 VAR PERSISTENT
//Conveyors Incoming 2000 (Purple line)
//Transport   
//----------------------------------------P2130--------------------------------------------------------------
cfgP2130IntlksArry: ARRAY [0..15] OF ST_CfgEvents := [
   (Description := 'Exit PE/Downstream MTR status' , DeviceLabel := '' , OKState := TRUE),   //DeviceLabel: Exit PE downstream
   (Description := 'System Interlocks' , DeviceLabel := '', OKState := TRUE, StopCode := E_StopCodes.SystemStop),
   13(())];
cfgP2130EvntsArry: ARRAY [0..15] OF ST_CfgEvents := [
   (Description := 'Jam Detected', DeviceLabel := '', LatchRequired := TRUE, OKState := FALSE, StopCode := E_StopCodes.ProductJam),   //DeviceLabel: Jam PE
   (),
   (Description := 'Disconnect', DeviceLabel := 'P2130', OKState := TRUE, StopCode := E_StopCodes.DisconnectState),   //DeviceLabel: Motor Disconnect
   (Description := 'System Fault', DeviceLabel := '', OKState := TRUE, FaultWarn:= TRUE, StopCode := E_StopCodes.SystemStop),
   (Description := 'RIO12182 Comm Fault', DeviceLabel := 'RIO12182', OKState := TRUE, FaultWarn:= TRUE, StopCode := E_StopCodes.FieldIOFLT),
   (Description := 'Power Transfer Raised', DeviceLabel := 'PX12151', OKState := TRUE, FaultWarn:= TRUE, StopCode := E_StopCodes.TransferLP),
   (Description := 'Motor Faulted', DeviceLabel := 'P2130', OKState := FALSE, StopCode := E_StopCodes.MotorOL),
   9(())];
//Transport
//----------------------------------------P2135--------------------------------------------------------------
cfgP2135IntlksArry: ARRAY [0..15] OF ST_CfgEvents := [
   (Description := 'Exit PE/Downstream MTR status' , DeviceLabel := '' , OKState := TRUE),   //DeviceLabel: Exit PE downstream
   (Description := 'System Interlocks' , DeviceLabel := '', OKState := TRUE, StopCode := E_StopCodes.SystemStop),
   11(())];
cfgP2135EvntsArry: ARRAY [0..15] OF ST_CfgEvents := [
   (Description := 'Jam Detected', DeviceLabel := '', LatchRequired := TRUE, OKState := FALSE, StopCode := E_StopCodes.ProductJam),   //DeviceLabel: Jam PE
   (),
   (Description := 'Disconnect', DeviceLabel := 'P2135', OKState := TRUE, StopCode := E_StopCodes.DisconnectState),   //DeviceLabel: Motor Disconnect
   (Description := 'System Fault', DeviceLabel := '', OKState := TRUE, FaultWarn:= TRUE, StopCode := E_StopCodes.SystemStop),
   (Description := 'RIO10161 Comm Fault', DeviceLabel := 'RIO10161', OKState := TRUE, FaultWarn:= TRUE, StopCode := E_StopCodes.FieldIOFLT),
   (Description := 'Motor Faulted', DeviceLabel := 'P2135', OKState := FALSE, StopCode := E_StopCodes.MotorOL),
   10(())];
//Transport
//----------------------------------------P2140--------------------------------------------------------------
cfgP2140IntlksArry: ARRAY [0..15] OF ST_CfgEvents := [
   (Description := 'Exit PE/Downstream MTR status' , DeviceLabel := '' , OKState := TRUE),   //DeviceLabel: Exit PE downstream
   (Description := 'System Interlocks' , DeviceLabel := '', OKState := TRUE, StopCode := E_StopCodes.SystemStop),
   (),
   (Description := 'GR2140-01 Auto', DeviceLabel := 'GR2140-01', OKState := TRUE, StopCode := E_StopCodes.DeviceNoInAuto),
   (Description := 'GR2140-02 Auto', DeviceLabel := 'GR2140-02', OKState := TRUE, StopCode := E_StopCodes.DeviceNoInAuto),
   (Description := 'PI2140-01 Auto', DeviceLabel := 'PI2140-01', OKState := TRUE, StopCode := E_StopCodes.DeviceNoInAuto),
   (Description := 'PL2140-01 Auto', DeviceLabel := 'PU2140-01', OKState := TRUE, StopCode := E_StopCodes.DeviceNoInAuto),
   9(())];
cfgP2140EvntsArry: ARRAY [0..15] OF ST_CfgEvents := [
   (Description := 'Jam Detected', DeviceLabel := '', LatchRequired := TRUE, OKState := FALSE, StopCode := E_StopCodes.ProductJam),   //DeviceLabel: Jam PE
   (),
   (Description := 'Disconnect', DeviceLabel := 'P2140', OKState := TRUE, StopCode := E_StopCodes.DisconnectState),   //DeviceLabel: Motor Disconnect
   (Description := 'System Fault', DeviceLabel := '', OKState := TRUE, FaultWarn:= TRUE, StopCode := E_StopCodes.SystemStop),
   (Description := 'RIO10161 Comm Fault', DeviceLabel := 'RIO10161', OKState := TRUE, FaultWarn:= TRUE, StopCode := E_StopCodes.FieldIOFLT),
   (Description := 'BCR_S2140_01 Comm Fault', DeviceLabel := 'BCR_S2140_01', OKState := TRUE, FaultWarn:= TRUE, StopCode := E_StopCodes.FieldIOFLT),
   (Description := 'Plow Jam', DeviceLabel := 'PL2140_01', OKState := TRUE, FaultWarn:= TRUE, StopCode := E_StopCodes.ProductJam),
   (Description := 'Motor Faulted', DeviceLabel := 'P2140', OKState := FALSE, StopCode := E_StopCodes.MotorOL),
   8(())];
//Transport
//----------------------------------------P2143--------------------------------------------------------------
cfgP2143IntlksArry: ARRAY [0..15] OF ST_CfgEvents := [
   (Description := 'Exit PE/Downstream MTR status' , DeviceLabel := '' , OKState := TRUE),   //DeviceLabel: Exit PE downstream
   (Description := 'System Interlocks' , DeviceLabel := '', OKState := TRUE, StopCode := E_StopCodes.SystemStop),
   13(())];
cfgP2143EvntsArry: ARRAY [0..15] OF ST_CfgEvents := [
   (Description := 'Jam Detected', DeviceLabel := '', LatchRequired := TRUE, OKState := FALSE, StopCode := E_StopCodes.ProductJam),   //DeviceLabel: Jam PE
   (),
   (Description := 'Disconnect', DeviceLabel := 'P2143', OKState := TRUE, StopCode := E_StopCodes.DisconnectState),   //DeviceLabel: Motor Disconnect
   (Description := 'System Fault', DeviceLabel := '', OKState := TRUE, FaultWarn:= TRUE, StopCode := E_StopCodes.SystemStop),
   (Description := 'RIO8171 Comm Fault', DeviceLabel := 'RIO8171', OKState := TRUE, FaultWarn:= TRUE, StopCode := E_StopCodes.FieldIOFLT),
   (Description := 'BCR_S2141_01 Comm Fault', DeviceLabel := 'BCR_S2141_011', OKState := TRUE, FaultWarn:= TRUE, StopCode := E_StopCodes.FieldIOFLT),
   (Description := 'Motor Faulted', DeviceLabel := 'P2143', OKState := FALSE, StopCode := E_StopCodes.MotorOL),
   9(())];
//Spiral
//----------------------------------------P2141--------------------------------------------------------------
cfgP2141IntlksArry: ARRAY [0..15] OF ST_CfgEvents := [
   (Description := 'Exit PE/Downstream MTR status' , DeviceLabel := '' , OKState := TRUE),   //DeviceLabel: Exit PE downstream
   (Description := 'System Interlocks' , DeviceLabel := '', OKState := TRUE, StopCode := E_StopCodes.SystemStop),
   14(())];
cfgP2141EvntsArry: ARRAY [0..15] OF ST_CfgEvents := [
   (Description := 'Jam Detected', DeviceLabel := '', LatchRequired := TRUE, OKState := FALSE, StopCode := E_StopCodes.ProductJam),   //DeviceLabel: Jam PE
   (),
   (Description := 'Disconnect', DeviceLabel := 'P2141', OKState := TRUE, StopCode := E_StopCodes.DisconnectState),   //DeviceLabel: Motor Disconnect
   (Description := 'System Fault', DeviceLabel := '', OKState := TRUE, FaultWarn:= TRUE, StopCode := E_StopCodes.SystemStop),
   (Description := 'RIO8171 Comm Fault', DeviceLabel := 'RIO8171', OKState := TRUE, FaultWarn:= TRUE, StopCode := E_StopCodes.FieldIOFLT),
   (Description := 'VFD State Not OK', DeviceLabel := 'P2141', OKState := TRUE, StopCode := E_StopCodes.VFD_Fault),
   10(())];
//Transport
//----------------------------------------P2142--------------------------------------------------------------
cfgP2142IntlksArry: ARRAY [0..15] OF ST_CfgEvents := [
   (Description := 'Exit PE/Downstream MTR status' , DeviceLabel := '' , OKState := TRUE),   //DeviceLabel: Exit PE downstream
   (Description := 'System Interlocks' , DeviceLabel := '', OKState := TRUE, StopCode := E_StopCodes.SystemStop),
   13(())];
cfgP2142EvntsArry: ARRAY [0..15] OF ST_CfgEvents := [
   (Description := 'Jam Detected', DeviceLabel := '', LatchRequired := TRUE, OKState := FALSE, StopCode := E_StopCodes.ProductJam),   //DeviceLabel: Jam PE
   (),
   (Description := 'Disconnect', DeviceLabel := 'P2142', OKState := TRUE, StopCode := E_StopCodes.DisconnectState),   //DeviceLabel: Motor Disconnect
   (Description := 'System Fault', DeviceLabel := '', OKState := TRUE, FaultWarn:= TRUE, StopCode := E_StopCodes.SystemStop),
   (Description := 'RIO8171 Comm Fault', DeviceLabel := 'RIO8171', OKState := TRUE, FaultWarn:= TRUE, StopCode := E_StopCodes.FieldIOFLT),
   (Description := 'Motor Faulted', DeviceLabel := 'P2142', OKState := FALSE, StopCode := E_StopCodes.MotorOL),
   10(())];
//Transport
//----------------------------------------P2145--------------------------------------------------------------
cfgP2145IntlksArry: ARRAY [0..15] OF ST_CfgEvents := [
   (Description := 'Exit PE/Downstream MTR status' , DeviceLabel := '' , OKState := TRUE),   //DeviceLabel: Exit PE downstream
   (Description := 'System Interlocks' , DeviceLabel := '', OKState := TRUE, StopCode := E_StopCodes.SystemStop),
   13(())];
cfgP2145EvntsArry: ARRAY [0..15] OF ST_CfgEvents := [
   (Description := 'Jam Detected', DeviceLabel := '', LatchRequired := TRUE, OKState := FALSE, StopCode := E_StopCodes.ProductJam),   //DeviceLabel: Jam PE
   (),
   (Description := 'Disconnect', DeviceLabel := 'P2145', OKState := TRUE, StopCode := E_StopCodes.DisconnectState),   //DeviceLabel: Motor Disconnect
   (Description := 'System Fault', DeviceLabel := '', OKState := TRUE, FaultWarn:= TRUE, StopCode := E_StopCodes.SystemStop),
   (Description := 'RIO2151 Comm Fault', DeviceLabel := 'RIO2151', OKState := TRUE, FaultWarn:= TRUE, StopCode := E_StopCodes.FieldIOFLT),
   (Description := 'Motor Faulted', DeviceLabel := 'P2145', OKState := FALSE, StopCode := E_StopCodes.MotorOL),
   10(())];
//Spiral
//----------------------------------------P2146--------------------------------------------------------------
cfgP2146IntlksArry: ARRAY [0..15] OF ST_CfgEvents := [
   (Description := 'Exit PE/Downstream MTR status' , DeviceLabel := '' , OKState := TRUE),   //DeviceLabel: Exit PE downstream
   (Description := 'System Interlocks' , DeviceLabel := '', OKState := TRUE, StopCode := E_StopCodes.SystemStop),
   (),
   12(())];
cfgP2146EvntsArry: ARRAY [0..15] OF ST_CfgEvents := [
   (Description := 'Jam Detected', DeviceLabel := '', LatchRequired := TRUE, OKState := FALSE, StopCode := E_StopCodes.ProductJam),   //DeviceLabel: Jam PE
   (),
   (Description := 'Disconnect', DeviceLabel := 'P2146', OKState := TRUE, StopCode := E_StopCodes.DisconnectState),   //DeviceLabel: Motor Disconnect
   (Description := 'System Fault', DeviceLabel := '', OKState := TRUE, FaultWarn:= TRUE, StopCode := E_StopCodes.SystemStop),
   (Description := 'RIO2151 Comm Fault', DeviceLabel := 'RIO2151', OKState := TRUE, FaultWarn:= TRUE, StopCode := E_StopCodes.FieldIOFLT),
   (Description := 'VFD State Not OK', DeviceLabel := 'P2146', OKState := TRUE, StopCode := E_StopCodes.VFD_Fault),
   10(())];
//Sorter
//----------------------------------------P2150--------------------------------------------------------------
cfgP2150IntlksArry: ARRAY [0..15] OF ST_CfgEvents := [
   (Description := 'Exit PE/Downstream MTR status' , DeviceLabel := '' , OKState := TRUE),   //DeviceLabel: Exit PE downstream
   (Description := 'System Interlocks' , DeviceLabel := '', OKState := TRUE, StopCode := E_StopCodes.SystemStop),
   (),
   (Description := 'GR2150-01 Auto', DeviceLabel := 'GR2150-01', OKState := TRUE, StopCode := E_StopCodes.DeviceNoInAuto),
   (Description := 'GR2150-02 Auto', DeviceLabel := 'GR2150-02', OKState := TRUE, StopCode := E_StopCodes.DeviceNoInAuto),
   (Description := 'PU2150-01 Auto', DeviceLabel := 'PU2150-01', OKState := TRUE, StopCode := E_StopCodes.DeviceNoInAuto),
   (Description := 'PU2150-02 Auto', DeviceLabel := 'PU2150-02', OKState := TRUE, StopCode := E_StopCodes.DeviceNoInAuto),
   (Description := 'PU2150-03 Auto', DeviceLabel := 'PU2150-03', OKState := TRUE, StopCode := E_StopCodes.DeviceNoInAuto),
   (Description := 'PU2150-04 Auto', DeviceLabel := 'PU2150-04', OKState := TRUE, StopCode := E_StopCodes.DeviceNoInAuto),
   7(())];
cfgP2150EvntsArry: ARRAY [0..15] OF ST_CfgEvents := [
   (Description := 'Jam Detected', DeviceLabel := '', LatchRequired := TRUE, OKState := FALSE, StopCode := E_StopCodes.ProductJam),   //DeviceLabel: Jam PE
   (),
   (Description := 'Disconnect', DeviceLabel := 'P2150', OKState := TRUE, StopCode := E_StopCodes.DisconnectState),   //DeviceLabel: Motor Disconnect
   (Description := 'System Fault', DeviceLabel := '', OKState := TRUE, FaultWarn:= TRUE, StopCode := E_StopCodes.SystemStop),
   (Description := 'RIO2151 Comm Fault', DeviceLabel := 'RIO2151', OKState := TRUE, FaultWarn:= TRUE, StopCode := E_StopCodes.FieldIOFLT),
   (Description := 'RIO3171 Comm Fault', DeviceLabel := 'RIO3171', OKState := TRUE, FaultWarn:= TRUE, StopCode := E_StopCodes.FieldIOFLT),
   (Description := 'RIO4141 Comm Fault', DeviceLabel := 'RIO4141', OKState := TRUE, FaultWarn:= TRUE, StopCode := E_StopCodes.FieldIOFLT),
   (Description := 'BCR_S2150_01 Comm Fault', DeviceLabel := 'BCR_S2150_01', OKState := TRUE, FaultWarn:= TRUE, StopCode := E_StopCodes.FieldIOFLT),
   (Description := 'Motor Faulted', DeviceLabel := 'P2150', OKState := FALSE, StopCode := E_StopCodes.MotorRunTO),
   7(())];
//Conveyors Incoming 3000 (Green line)
//Spiral
//----------------------------------------P3080--------------------------------------------------------------
cfgP3080IntlksArry: ARRAY [0..15] OF ST_CfgEvents := [
   (Description := 'Exit PE/Downstream MTR status' , DeviceLabel := '' , OKState := TRUE),   //DeviceLabel: Exit PE downstream
   (Description := 'System Interlocks' , DeviceLabel := '', OKState := TRUE, StopCode := E_StopCodes.SystemStop),
   (),
   12(())];
cfgP3080EvntsArry: ARRAY [0..15] OF ST_CfgEvents := [
   (Description := 'Jam Detected', DeviceLabel := '', LatchRequired := TRUE, OKState := FALSE, StopCode := E_StopCodes.ProductJam),   //DeviceLabel: Jam PE
   (),
   (Description := 'Disconnect', DeviceLabel := 'P3080', OKState := TRUE, StopCode := E_StopCodes.DisconnectState),   //DeviceLabel: Motor Disconnect
   (Description := 'System Fault', DeviceLabel := '', OKState := TRUE, FaultWarn:= TRUE, StopCode := E_StopCodes.SystemStop),
   (Description := 'RIO9191 Comm Fault', DeviceLabel := 'RIO9191', OKState := TRUE, FaultWarn:= TRUE, StopCode := E_StopCodes.FieldIOFLT),
   (Description := 'BCR_S2150_01 Comm Fault', DeviceLabel := 'BCR_S2150_01', OKState := TRUE, FaultWarn:= TRUE, StopCode := E_StopCodes.FieldIOFLT),
   (Description := 'Height Check', DeviceLabel := 'PE_12261', OKState := TRUE, FaultWarn:= TRUE, StopCode := E_StopCodes.OverHeightFLT),
   (Description := 'VFD State Not OK', DeviceLabel := 'P3080', OKState := TRUE, StopCode := E_StopCodes.VFD_Fault),
   8(())];
//Transport
//----------------------------------------P3085--------------------------------------------------------------
cfgP3085IntlksArry: ARRAY [0..15] OF ST_CfgEvents := [
   (Description := 'Exit PE/Downstream MTR status' , DeviceLabel := '' , OKState := TRUE),   //DeviceLabel: Exit PE downstream
   (Description := 'System Interlocks' , DeviceLabel := '', OKState := TRUE, StopCode := E_StopCodes.SystemStop),
   (),
   12(())];
cfgP3085EvntsArry: ARRAY [0..15] OF ST_CfgEvents := [
   (Description := 'Jam Detected', DeviceLabel := '', LatchRequired := TRUE, OKState := FALSE, StopCode := E_StopCodes.ProductJam),   //DeviceLabel: Jam PE
   (),
   (Description := 'Disconnect', DeviceLabel := 'P3085', OKState := TRUE, StopCode := E_StopCodes.DisconnectState),   //DeviceLabel: Motor Disconnect
   (Description := 'System Fault', DeviceLabel := '', OKState := TRUE, FaultWarn:= TRUE, StopCode := E_StopCodes.SystemStop),
   (Description := 'RIO12182 Comm Fault', DeviceLabel := 'RIO12182', OKState := TRUE, FaultWarn:= TRUE, StopCode := E_StopCodes.FieldIOFLT),
   (Description := 'Motor Faulted', DeviceLabel := 'P3085', OKState := FALSE, StopCode := E_StopCodes.MotorRunTO),
   10(())];
//Transport
//----------------------------------------P3090--------------------------------------------------------------
cfgP3090IntlksArry: ARRAY [0..15] OF ST_CfgEvents := [
   (Description := 'Exit PE/Downstream MTR status' , DeviceLabel := '' , OKState := TRUE),   //DeviceLabel: Exit PE downstream
   (Description := 'System Interlocks' , DeviceLabel := '', OKState := TRUE, StopCode := E_StopCodes.SystemStop),
   (),
   12(())];
cfgP3090EvntsArry: ARRAY [0..15] OF ST_CfgEvents := [
   (Description := 'Jam Detected', DeviceLabel := '', LatchRequired := TRUE, OKState := FALSE, StopCode := E_StopCodes.ProductJam),   //DeviceLabel: Jam PE
   (),
   (Description := 'Disconnect', DeviceLabel := 'P3090', OKState := TRUE, StopCode := E_StopCodes.DisconnectState),   //DeviceLabel: Motor Disconnect
   (Description := 'System Fault', DeviceLabel := '', OKState := TRUE, FaultWarn:= TRUE, StopCode := E_StopCodes.SystemStop),
   (Description := 'RIO12182 Comm Fault', DeviceLabel := 'RIO12182', OKState := TRUE, FaultWarn:= TRUE, StopCode := E_StopCodes.FieldIOFLT),
   (Description := 'Motor Faulted', DeviceLabel := 'P3090', OKState := FALSE, StopCode := E_StopCodes.MotorRunTO),
   10(())];
//Transport
//----------------------------------------P3095--------------------------------------------------------------
cfgP3095IntlksArry: ARRAY [0..15] OF ST_CfgEvents := [
   (Description := 'Exit PE/Downstream MTR status' , DeviceLabel := '' , OKState := TRUE),   //DeviceLabel: Exit PE downstream
   (Description := 'System Interlocks' , DeviceLabel := '', OKState := TRUE, StopCode := E_StopCodes.SystemStop),
   (),
   12(())];
cfgP3095EvntsArry: ARRAY [0..15] OF ST_CfgEvents := [
   (Description := 'Jam Detected', DeviceLabel := '', LatchRequired := TRUE, OKState := FALSE, StopCode := E_StopCodes.ProductJam),   //DeviceLabel: Jam PE
   (),
   (Description := 'Disconnect', DeviceLabel := 'P3095', OKState := TRUE, StopCode := E_StopCodes.DisconnectState),   //DeviceLabel: Motor Disconnect
   (Description := 'System Fault', DeviceLabel := '', OKState := TRUE, FaultWarn:= TRUE, StopCode := E_StopCodes.SystemStop),
   (Description := 'RIO12182 Comm Fault', DeviceLabel := 'RIO12182', OKState := TRUE, FaultWarn:= TRUE, StopCode := E_StopCodes.FieldIOFLT),
   (Description := 'Power Transfer Raised', DeviceLabel := 'PX12251', OKState := TRUE, FaultWarn:= TRUE, StopCode := E_StopCodes.TransferLP),
   (Description := 'Motor Faulted', DeviceLabel := 'P3095', OKState := FALSE, StopCode := E_StopCodes.MotorOL),
   9(())];
P2141_Velocity: INT := 1800;
P2146_Velocity: INT := 1800;
P3080_Velocity: INT := 1800;
END_VAR

ResetAllDrives := System.Cnvyr_Reset; //Reset For VFD
//EAP
GVL_IO.To205_P2130_IsRunning := P2130_Status.Sts_IsRunning;
GVL_IO.To205_P3095_SendingProduct := P3095_Status.Sts_IsRunning OR Photoeyes.PE_12091.Out OR Photoeyes.PE_12181.Out;

//Conveyors Incoming 2000 (Purple line)
//Transport
//----------------------------------------P2130--------------------------------------------------------------
P2130_StatePB.AutoPB := System.Cnvyr_Auto;
P2130_StatePB.ManPB := System.Cnvyr_Manual;
P2130_StatePB.ResetPB := System.Cnvyr_Reset;
P2130_StatePB.OfflinePB := System.Cnvyr_Offline;
P2130SleepWakeTrig[1] := GVL_IO.From205_P2125_SendingProduct; //EAP Wakeup bits 

// Initialize the Equipment Type
P2130_Status.Sts_EquipmentState.EquipType := E_EquipType.Conveyor;

// Interlocks
//P2130.In_EquipIntlks.2:=
//Events
P2130.In_EquipEvents.2:= GVL_IO.DS_P2130;
P2130.In_EquipEvents.3:= System.SysEventsAllOk;
P2130.In_EquipEvents.4:= NOT CommStatus.RIO12182_CommFault.Out;
P2130.In_EquipEvents.5:= ProxSensors.PX_12151_Extended.Out;
P2130.In_EquipEvents.6:= NOT GVL_IO.P2130_Faulted;

// Function Call
P2130(
   In_p_EquipStatePB:= P2130_StatePB,
   In_P_ConvReqRun:= TRUE,
   In_ConvDwnStrmMtrStatus:=  P2135_Status.Sts_IsRunning,
   In_ConvCrntExitPhotoEye:=  Photoeyes.PE_12171.Out,
   In_SimActive:= System.Sys_SimActive,
   In_EquipInit:= GVL_IO.INIT,
   In_WakeSlpTrigArry:= P2130SleepWakeTrig,
   Cfg_EquipIndex := GVL_EquipArrays.nEquipIndex,
   Cfg_EquipLabel := cfgP2130Label,
   Cfg_EquipDefState:= System.ConvDefaultState,
   Cfg_EquipIntlksArry:= cfgP2130IntlksArry,
   Cfg_EquipEvntsArry:= cfgP2130EvntsArry,
   cfg_JamDetectTime:= cfgP2130JamDetectTime,
   Cfg_UseSleepTmr := TRUE,
   Cfg_UseStartUpDelay := TRUE,
   Cfg_StartUpDelayTime := T#500MS,
   Cfg_SleepWaitTime:= cfgP2130SleepTime,
   Sts_EquipState := P2130_Status,
   Out_ConvCrntMtr => GVL_IO.P2130_RUN);

P2130_Status.Sts_IsRunning := GVL_IO.P2130_RUN;

//Transport
//----------------------------------------P2135--------------------------------------------------------------
P2135_StatePB.AutoPB := System.Cnvyr_Auto;
P2135_StatePB.ManPB := System.Cnvyr_Manual;
P2135_StatePB.ResetPB := System.Cnvyr_Reset;
P2135_StatePB.OfflinePB := System.Cnvyr_Offline;
P2135SleepWakeTrig[1] := Photoeyes.PE_12171.Out;
//EAP from 3rd floor

// Initialize the Equipment Type
P2135_Status.Sts_EquipmentState.EquipType := E_EquipType.Conveyor;

// Interlocks
//P2135.In_EquipIntlks.2:=
//Events
P2135.In_EquipEvents.2:= GVL_IO.DS_P2135;
P2135.In_EquipEvents.3:= System.SysEventsAllOk;
P2135.In_EquipEvents.4:= NOT CommStatus.RIO10161_CommFault.Out;
P2135.In_EquipEvents.5:= NOT GVL_IO.P2135_Faulted;

// Function Call
P2135(
   In_p_EquipStatePB:= P2135_StatePB,
   In_P_ConvReqRun:= TRUE,
   In_ConvDwnStrmMtrStatus:= P2140_Status.Sts_IsRunning,
   In_ConvCrntExitPhotoEye:=  Photoeyes.PE_10291.Out,
   In_SimActive:= System.Sys_SimActive,
   In_EquipInit:= GVL_IO.INIT,
   In_WakeSlpTrigArry:= P2135SleepWakeTrig,
   Cfg_EquipIndex := GVL_EquipArrays.nEquipIndex,
   Cfg_EquipLabel := cfgP2135Label,
   Cfg_EquipDefState:= System.ConvDefaultState,
   Cfg_EquipIntlksArry:= cfgP2135IntlksArry,
   Cfg_EquipEvntsArry:= cfgP2135EvntsArry,
   cfg_JamDetectTime:= cfgP2135JamDetectTime,
   Cfg_UseSleepTmr := TRUE,
   Cfg_UseStartUpDelay := TRUE,
   Cfg_StartUpDelayTime := T#500MS,
   Cfg_SleepWaitTime:= cfgP2135SleepTime,
   Sts_EquipState := P2135_Status,
   Out_ConvCrntMtr => GVL_IO.P2135_RUN);

P2135_Status.Sts_IsRunning := GVL_IO.P2135_RUN;
//Transport
//----------------------------------------P2140--------------------------------------------------------------
P2140_StatePB.AutoPB := System.Cnvyr_Auto;
P2140_StatePB.ManPB := System.Cnvyr_Manual;
P2140_StatePB.ResetPB := System.Cnvyr_Reset;
P2140_StatePB.OfflinePB := System.Cnvyr_Offline;
P2140SleepWakeTrig[1] := Photoeyes.PE_10291.Out;
P2140SleepWakeTrig[2] := Photoeyes.PE_12171.Out;

// Initialize the Equipment Type
P2140_Status.Sts_EquipmentState.EquipType := E_EquipType.Conveyor;

// Interlocks
P2140.In_EquipIntlks.3:= Solenoids.GR2140_01_Status.Sts_EquipmentState.StsAuto;
P2140.In_EquipIntlks.4:= Solenoids.GR2140_02_Status.Sts_EquipmentState.StsAuto;
P2140.In_EquipIntlks.5:= Solenoids.PI2140_01_Status.Sts_EquipmentState.StsAuto;
P2140.In_EquipIntlks.6:= Solenoids.PL2140_01_Status.Sts_EquipmentState.StsAuto; 
//Events
P2140.In_EquipEvents.2:= GVL_IO.DS_P2140;
P2140.In_EquipEvents.3:= System.SysEventsAllOk;
P2140.In_EquipEvents.4:= NOT CommStatus.RIO10161_CommFault.Out;
P2140.In_EquipEvents.5:= NOT CommStatus.BCR_S2140_01_CommFault.Out;
P2140.In_EquipEvents.6:= FALSE;//Photoeyes.PE_10151.JamDetected AND Not Solenoids.PL2140_01.Out_ExtendCrntSV;
P2140.In_EquipEvents.7:= NOT GVL_IO.P2140_Faulted;
P2140.In_EquipEvents.8:= Photoeyes.PE_10151.JamDetected; 

// Function Call
P2140(
   In_p_EquipStatePB:= P2140_StatePB,
   In_P_ConvReqRun:= TRUE,
   In_ConvDwnStrmMtrStatus:= P2145_Status.Sts_IsRunning,
   In_ConvCrntExitPhotoEye:= Photoeyes.PE_10091.Out,
   In_SimActive:= System.Sys_SimActive,
   In_EquipInit:= GVL_IO.INIT,
   In_WakeSlpTrigArry:= P2140SleepWakeTrig,
   Cfg_EquipIndex := GVL_EquipArrays.nEquipIndex,
   Cfg_EquipLabel := cfgP2140Label,
   Cfg_EquipDefState:= System.ConvDefaultState,
   Cfg_EquipIntlksArry:= cfgP2140IntlksArry,
   Cfg_EquipEvntsArry:= cfgP2140EvntsArry,
   cfg_JamDetectTime:= cfgP2140JamDetectTime,
   Cfg_UseSleepTmr := TRUE,
   Cfg_UseStartUpDelay := TRUE,
   Cfg_StartUpDelayTime := T#500MS,
   Cfg_SleepWaitTime:= cfgP2140SleepTime,
   Sts_EquipState := P2140_Status,
   Out_ConvCrntMtr => GVL_IO.P2140_RUN);

P2140_Status.Sts_IsRunning := GVL_IO.P2140_RUN;
//Transport
//----------------------------------------P2143--------------------------------------------------------------
P2143_StatePB.AutoPB := System.Cnvyr_Auto;
P2143_StatePB.ManPB := System.Cnvyr_Manual;
P2143_StatePB.ResetPB := System.Cnvyr_Reset;
P2143_StatePB.OfflinePB := System.Cnvyr_Offline;
P2143SleepWakeTrig[1] := Photoeyes.PE_10291.Out;
P2143SleepWakeTrig[2] := Photoeyes.PE_12171.Out;

// Initialize the Equipment Type
P2143_Status.Sts_EquipmentState.EquipType := E_EquipType.Conveyor;

// Interlocks
//P2143.In_EquipIntlks.2:= 
//Events
P2143.In_EquipEvents.2:= GVL_IO.DS_P2143;
P2143.In_EquipEvents.3:= System.SysEventsAllOk;
P2143.In_EquipEvents.4:= NOT CommStatus.RIO8171_CommFault.Out;
P2143.In_EquipEvents.5:= NOT CommStatus.BCR_S2141_01_CommFault.Out;
P2143.In_EquipEvents.6:= NOT GVL_IO.P2143_Faulted;

// Function Call
P2143(
   In_p_EquipStatePB:= P2143_StatePB,
   In_P_ConvReqRun:= TRUE,
   In_ConvDwnStrmMtrStatus:=  P2141_VFD.IsRunning,
   In_ConvCrntExitPhotoEye:= Photoeyes.PE_8161.Out,
   In_SimActive:= System.Sys_SimActive,
   In_EquipInit:= GVL_IO.INIT,
   In_WakeSlpTrigArry:= P2143SleepWakeTrig,
   Cfg_EquipIndex := GVL_EquipArrays.nEquipIndex,
   Cfg_EquipLabel := cfgP2143Label,
   Cfg_EquipDefState:= System.ConvDefaultState,
   Cfg_EquipIntlksArry:= cfgP2143IntlksArry,
   Cfg_EquipEvntsArry:= cfgP2143EvntsArry,
   cfg_JamDetectTime:= cfgP2143JamDetectTime,
   Cfg_UseSleepTmr := TRUE,
   Cfg_UseStartUpDelay := TRUE,
   Cfg_StartUpDelayTime := T#500MS,
   Cfg_SleepWaitTime:= cfgP2143SleepTime,
   Sts_EquipState := P2143_Status,
   Out_ConvCrntMtr => GVL_IO.P2143_RUN);

P2143_Status.Sts_IsRunning := GVL_IO.P2143_RUN;
//Spiral
//----------------------------------------P2141--------------------------------------------------------------
P2141_StatePB.AutoPB := System.Cnvyr_Auto;
P2141_StatePB.ManPB := System.Cnvyr_Manual;
P2141_StatePB.ResetPB := System.Cnvyr_Reset;
P2141_StatePB.OfflinePB := System.Cnvyr_Offline;
P2141SleepWakeTrig[1] := Photoeyes.PE_8161.Out;
P2141SleepWakeTrig[2] := Photoeyes.PE_10151.Out;

// Initialize the Equipment Type
P2141_Status.Sts_EquipmentState.EquipType := E_EquipType.Conveyor;

// Interlocks
// Interlock the full for a stop only when the warning is on for the downstream conveyor
P2141.In_EquipIntlks.2:= Photoeyes.PE_8131.Out_OnOffFltrd AND P2142.Sts_WarnsArry[6].Status;

//Events
P2141.In_EquipEvents.2:= GVL_IO.DS_P2141;
P2141.In_EquipEvents.3:= System.SysEventsAllOk;
P2141.In_EquipEvents.4:= NOT CommStatus.RIO8171_CommFault.Out;
P2141.In_EquipEvents.5:= NOT P2141_VFD.IsFaulted;

// Function Call
P2141(
   In_p_EquipStatePB:= P2141_StatePB,
   In_P_ConvReqRun:= TRUE,
   In_ConvDwnStrmMtrStatus:= P2142_Status.Sts_IsRunning AND NOT P2142.Sts_WarnsArry[6].Status,
   In_ConvCrntExitPhotoEye:= Photoeyes.PE_8131.Out,
   In_SimActive:= System.Sys_SimActive,
   In_EquipInit:= GVL_IO.INIT,
   In_WakeSlpTrigArry:= P2141SleepWakeTrig,
   Cfg_EquipIndex := GVL_EquipArrays.nEquipIndex,
   Cfg_EquipLabel := cfgP2141Label,
   Cfg_EquipDefState:= System.ConvDefaultState,
   Cfg_EquipIntlksArry:= cfgP2141IntlksArry,
   Cfg_EquipEvntsArry:= cfgP2141EvntsArry,
   cfg_JamDetectTime:= cfgP2141JamDetectTime,
   Cfg_UseSleepTmr := TRUE,
   Cfg_UseStartUpDelay := TRUE,
   Cfg_StartUpDelayTime := T#500MS,
   Cfg_SleepWaitTime:= cfgP2141SleepTime,
   Sts_EquipState := P2141_Status);

//Motor Control
P2141_VFD(
   RunVelocity := P2141_Velocity,
   VelocityThreshold := DefaultVelocityThreshold,
   Reset := ResetAllDrives,
   RunRequest := (P2141.Out_ConvCrntMtr OR Test_VFD_P2141));
P2141_Status.Sts_IsRunning := P2141_VFD.IsRunning;
//Transport
//----------------------------------------P2142--------------------------------------------------------------
P2142_StatePB.AutoPB := System.Cnvyr_Auto;
P2142_StatePB.ManPB := System.Cnvyr_Manual;
P2142_StatePB.ResetPB := System.Cnvyr_Reset;
P2142_StatePB.OfflinePB := System.Cnvyr_Offline;
P2142SleepWakeTrig[1] := Photoeyes.PE_8131.Out;
P2142SleepWakeTrig[2] := Photoeyes.PE_8161.Out;

// Initialize the Equipment Type
P2142_Status.Sts_EquipmentState.EquipType := E_EquipType.Conveyor;

// Interlocks
//P2142.In_EquipIntlks.2:= Photoeyes.PE_8141.Out_OnFltrd;

//Events
P2142.In_EquipEvents.2:= GVL_IO.DS_P2142;
P2142.In_EquipEvents.3:= System.SysEventsAllOk;
P2142.In_EquipEvents.4:= NOT CommStatus.RIO8171_CommFault.Out;
P2142.In_EquipEvents.5:= NOT GVL_IO.P2142_Faulted;
P2142.In_EquipEvents.6 := Photoeyes.PE_8141.Out_OnOffFltrd AND Photoeyes.PE_8191.Out_OnOffFltrd;

// Function Call
P2142(
   In_p_EquipStatePB:= P2142_StatePB,
   In_P_ConvReqRun:= TRUE,
   In_ConvDwnStrmMtrStatus:= TRUE,
   In_ConvCrntExitPhotoEye:=  FALSE,
   Cfg_ConvType:= E_ConvType.end,
   In_SimActive:= System.Sys_SimActive,
   In_EquipInit:= GVL_IO.INIT,
   In_WakeSlpTrigArry:= P2142SleepWakeTrig,
   Cfg_EquipIndex := GVL_EquipArrays.nEquipIndex,
   Cfg_EquipLabel := cfgP2142Label,
   Cfg_EquipDefState:= System.ConvDefaultState,
   Cfg_EquipIntlksArry:= cfgP2142IntlksArry,
   Cfg_EquipEvntsArry:= cfgP2142EvntsArry,
   cfg_JamDetectTime:= cfgP2142JamDetectTime,
   Cfg_UseSleepTmr := TRUE,
   Cfg_UseStartUpDelay := TRUE,
   Cfg_StartUpDelayTime := T#500MS,
   Cfg_SleepWaitTime:= cfgP2142SleepTime,
   Sts_EquipState := P2142_Status,
   Out_ConvCrntMtr => GVL_IO.P2142_RUN);

P2142_Status.Sts_IsRunning := GVL_IO.P2142_RUN;
//Transport
//----------------------------------------P2145--------------------------------------------------------------
P2145_StatePB.AutoPB := System.Cnvyr_Auto;
P2145_StatePB.ManPB := System.Cnvyr_Manual;
P2145_StatePB.ResetPB := System.Cnvyr_Reset;
P2145_StatePB.OfflinePB := System.Cnvyr_Offline;
P2145SleepWakeTrig[1] := PhotoEyes.PE_10091.Out_OffFltrd;
P2145SleepWakeTrig[2] := PhotoEyes.PE_10291.Out_OffFltrd;

// Initialize the Equipment Type
P2145_Status.Sts_EquipmentState.EquipType := E_EquipType.Conveyor;

// Interlocks
//P2145.In_EquipIntlks.2:= 
//Events
P2145.In_EquipEvents.2:= GVL_IO.DS_P2145;
P2145.In_EquipEvents.3:= System.SysEventsAllOk;
P2145.In_EquipEvents.4:= NOT CommStatus.RIO2151_CommFault.Out;
P2145.In_EquipEvents.5:= NOT GVL_IO.P2145_Faulted;

// Function Call
P2145(
   In_p_EquipStatePB:= P2145_StatePB,
   In_P_ConvReqRun:= TRUE,
   In_ConvDwnStrmMtrStatus:=  P2146_VFD.IsRunning,
   In_ConvCrntExitPhotoEye:=  PhotoEyes.PE_2231.Out,
   In_SimActive:= System.Sys_SimActive,
   In_EquipInit:= GVL_IO.INIT,
   In_WakeSlpTrigArry:= P2145SleepWakeTrig,
   Cfg_EquipIndex := GVL_EquipArrays.nEquipIndex,
   Cfg_EquipLabel := cfgP2145Label,
   Cfg_EquipDefState:= System.ConvDefaultState,
   Cfg_EquipIntlksArry:= cfgP2145IntlksArry,
   Cfg_EquipEvntsArry:= cfgP2145EvntsArry,
   cfg_JamDetectTime:= cfgP2145JamDetectTime,
   Cfg_UseSleepTmr := TRUE,
   Cfg_UseStartUpDelay := TRUE,
   Cfg_StartUpDelayTime := T#500MS,
   Cfg_SleepWaitTime:= cfgP2145SleepTime,
   Sts_EquipState := P2145_Status,
   Out_ConvCrntMtr => GVL_IO.P2145_RUN);

P2145_Status.Sts_IsRunning := GVL_IO.P2145_RUN;
//Spiral
//----------------------------------------P2146--------------------------------------------------------------
P2146_StatePB.AutoPB := System.Cnvyr_Auto;
P2146_StatePB.ManPB := System.Cnvyr_Manual;
P2146_StatePB.ResetPB := System.Cnvyr_Reset;
P2146_StatePB.OfflinePB := System.Cnvyr_Offline;
P2146SleepWakeTrig[1] := PhotoEyes.PE_2231.Out_OffFltrd;
P2145SleepWakeTrig[2] := PhotoEyes.PE_10091.Out_OffFltrd;

// Initialize the Equipment Type
P2146_Status.Sts_EquipmentState.EquipType := E_EquipType.Conveyor;

// Interlocks
P2146.In_EquipIntlks.2:= Photoeyes.PE_2101.Out_OnOffFltrd AND Photoeyes.PE_2201.Out_OnOffFltrd;
//Events
P2146.In_EquipEvents.2:= GVL_IO.DS_P2146;
P2146.In_EquipEvents.3:= System.SysEventsAllOk;
P2146.In_EquipEvents.4:= NOT CommStatus.RIO2151_CommFault.Out;
P2146.In_EquipEvents.5:= NOT P2146_VFD.IsFaulted;

// Function Call
P2146(
   In_p_EquipStatePB:= P2146_StatePB,
   In_P_ConvReqRun:= TRUE,
   In_ConvDwnStrmMtrStatus:= P2150_Status.Sts_IsRunning,
   In_ConvCrntExitPhotoEye:= Photoeyes.PE_2201.Out_OffFltrd,
   In_SimActive:= System.Sys_SimActive,
   In_EquipInit:= GVL_IO.INIT,
   In_WakeSlpTrigArry:= P2146SleepWakeTrig,
   Cfg_EquipIndex := GVL_EquipArrays.nEquipIndex,
   Cfg_EquipLabel := cfgP2146Label,
   Cfg_EquipDefState:= System.ConvDefaultState,
   Cfg_EquipIntlksArry:= cfgP2146IntlksArry,
   Cfg_EquipEvntsArry:= cfgP2146EvntsArry,
   cfg_JamDetectTime:= cfgP2146JamDetectTime,
   Cfg_UseSleepTmr := TRUE,
   Cfg_UseStartUpDelay := FALSE,
   Cfg_SleepWaitTime:= cfgP2146SleepTime,
   Sts_EquipState := P2146_Status);

//Motor Control
P2146_VFD(
   RunVelocity := P2146_Velocity,
   VelocityThreshold := DefaultVelocityThreshold,
   Reset := ResetAllDrives,
   RunRequest := (P2146.Out_ConvCrntMtr OR Test_VFD_P2146));
P2146_Status.Sts_IsRunning := P2146_VFD.IsRunning;
//Sorter
//----------------------------------------P2150--------------------------------------------------------------
P2150_StatePB.AutoPB := System.Cnvyr_Auto OR GVL_IO.PB_RemoteReset_3211;
P2150_StatePB.ManPB := System.Cnvyr_Manual;
P2150_StatePB.ResetPB := System.Cnvyr_Reset OR GVL_IO.PB_RemoteReset_3211;
P2150_StatePB.OfflinePB := System.Cnvyr_Offline;
P2150SleepWakeTrig[1] := PhotoEyes.PE_2201.Out_OffFltrd;
P2150SleepWakeTrig[2] := PhotoEyes.PE_2231.Out_OffFltrd;
P2150SleepWakeTrig[3] := PhotoEyes.PE_2131.Out_OffFltrd;
P2150SleepWakeTrig[4] := PhotoEyes.PE_2101.Out_OffFltrd;


// Initialize the Equipment Type
P2150_Status.Sts_EquipmentState.EquipType := E_EquipType.Conveyor;

// Interlocks
P2150.In_EquipIntlks.2:= Singulation_Control.SortSingulation_P2150.Out_Ready;
P2150.In_EquipIntlks.3:= Solenoids.GR2150_01_Status.Sts_EquipmentState.StsAuto;
P2150.In_EquipIntlks.4:= Solenoids.PI2150_01_Status.Sts_EquipmentState.StsAuto;
P2150.In_EquipIntlks.5:= Solenoids.PU2150_01_Status.Sts_EquipmentState.StsAuto;
P2150.In_EquipIntlks.6:= Solenoids.PU2150_02_Status.Sts_EquipmentState.StsAuto;
P2150.In_EquipIntlks.7:= Solenoids.PU2150_03_Status.Sts_EquipmentState.StsAuto;
P2150.In_EquipIntlks.8:= Solenoids.PU2150_04_Status.Sts_EquipmentState.StsAuto;
P2150.In_EquipIntlks.9:= Sorter.aSorterDiverts_P2150[1].Full;
P2150.In_EquipIntlks.10:= Sorter.aSorterDiverts_P2150[2].Full;
P2150.In_EquipIntlks.11:= Sorter.aSorterDiverts_P2150[3].Full;
P2150.In_EquipIntlks.12:= Sorter.aSorterDiverts_P2150[4].Full;

//Events
P2150.In_EquipEvents.2:= GVL_IO.DS_P2150;
P2150.In_EquipEvents.3:= System.SysEventsAllOk;
P2150.In_EquipEvents.4:= NOT CommStatus.RIO2151_CommFault.Out;
P2150.In_EquipEvents.5:= NOT CommStatus.RIO3171_CommFault.Out;
P2150.In_EquipEvents.6:= NOT CommStatus.RIO4141_CommFault.Out;
P2150.In_EquipEvents.7:= NOT CommStatus.BCR_S2150_01_CommFault.Out;
P2150.In_EquipEvents.8:= NOT GVL_IO.P2150_Faulted;
P2150.In_EquipEvents.9:= Photoeyes.PE_2101.Out_OnOffFltrd;
P2150.In_EquipEvents.10:= Sorter.aSorterDiverts_P2150[1].Jammed;
P2150.In_EquipEvents.11:= Sorter.aSorterDiverts_P2150[2].Jammed;
P2150.In_EquipEvents.12:= Sorter.aSorterDiverts_P2150[3].Jammed;
P2150.In_EquipEvents.13:= Sorter.aSorterDiverts_P2150[4].Jammed;

// Function Call
P2150(
	In_p_EquipStatePB:= P2150_StatePB,
	In_P_ConvReqRun:= TRUE,
	In_ConvCrntExitPhotoEye:= PhotoEyes.PE_4161.Out,
	Cfg_ConvType:= E_ConvType.end,
	In_SimActive:= System.Sys_SimActive,
	In_EquipInit:= GVL_IO.INIT,
	In_WakeSlpTrigArry:= P2150SleepWakeTrig,
	Cfg_EquipIndex := GVL_EquipArrays.nEquipIndex,
	Cfg_EquipLabel := cfgP2150Label,
	Cfg_EquipDefState:= System.ConvDefaultState,
	Cfg_EquipIntlksArry:= cfgP2150IntlksArry,
	Cfg_EquipEvntsArry:= cfgP2150EvntsArry,
	cfg_JamDetectTime:= T#2S,
	Cfg_UseSleepTmr := TRUE,
	Cfg_SleepWaitTime:= cfgP2150SleepTime,
	Sts_EquipState := P2150_Status,
	Out_ConvCrntMtr => GVL_IO.P2150_RUN);

P2150_Status.Sts_IsRunning := GVL_IO.P2150_RUN;
//Conveyors Incoming 3000 (Green line)
//Spiral
//----------------------------------------P3080--------------------------------------------------------------
P3080_StatePB.AutoPB := System.Cnvyr_Auto OR GVL_IO.PB_RemoteReset_8251;
P3080_StatePB.ManPB := System.Cnvyr_Manual;
P3080_StatePB.ResetPB := System.Cnvyr_Reset OR GVL_IO.PB_RemoteReset_8251;
P3080_StatePB.OfflinePB := System.Cnvyr_Offline;
P3080_ResetWakeTmr(IN:= GVL_IO.PB_RemoteReset_8251, PT:= T#3S, Q=> );
P3080SleepWakeTrig[1] := P3080_ResetWakeTmr.Q; //Reset Button
P3080SleepWakeTrig[2] := Photoeyes.PE_9141.Out; //Photo Eye
P3080SleepWakeTrig[3] := Photoeyes.PE_9161.Out; //Photo Eye
P3080SleepWakeTrig[4] := Photoeyes.PE_9191.Out; //Photo Eye

// Initialize the Equipment Type
P3080_Status.Sts_EquipmentState.EquipType := E_EquipType.Conveyor;

// Interlocks
//P3080.In_EquipIntlks.2:= 
//Events
P3080.In_EquipEvents.2:= GVL_IO.DS_P3080;
P3080.In_EquipEvents.3:= System.SysEventsAllOk;
P3080.In_EquipEvents.4:= NOT CommStatus.RIO9191_CommFault.Out;
P3080.In_EquipEvents.5:= NOT CommStatus.BCR_S2150_01_CommFault.Out;
P3080.In_EquipEvents.6:= Photoeyes.PE_9221.Out;
P3080.In_EquipEvents.7:= NOT P3080_VFD.IsFaulted;

// Function Call
P3080(
   In_p_EquipStatePB:= P3080_StatePB,
   In_P_ConvReqRun:= TRUE,
   In_ConvDwnStrmMtrStatus:= P3085_Status.Sts_IsRunning,
   In_ConvCrntExitPhotoEye:= Photoeyes.PE_9191.Out, 
   In_SimActive:= System.Sys_SimActive,
   In_EquipInit:= GVL_IO.INIT,
   In_WakeSlpTrigArry:= P3080SleepWakeTrig,
   Cfg_EquipIndex := GVL_EquipArrays.nEquipIndex,
   Cfg_EquipLabel := cfgP3080Label,
   Cfg_EquipDefState:= System.ConvDefaultState,
   Cfg_EquipIntlksArry:= cfgP3080IntlksArry,
   Cfg_EquipEvntsArry:= cfgP3080EvntsArry,
   cfg_JamDetectTime:= cfgP3080JamDetectTime,
   Cfg_UseSleepTmr := TRUE,
   Cfg_UseStartUpDelay := TRUE,
   Cfg_StartUpDelayTime := T#500MS,
   Cfg_SleepWaitTime:= cfgP3080SleepTime,
   Sts_EquipState := P3080_Status);

//Motor Control
P3080_VFD(
   RunVelocity := P3080_Velocity,
   VelocityThreshold := DefaultVelocityThreshold,
   Reset := ResetAllDrives,
   RunRequest := (P3080.Out_ConvCrntMtr OR Test_VFD_P3080));
P3080_Status.Sts_IsRunning := P3080_VFD.IsRunning;
//Transport
//----------------------------------------P3085--------------------------------------------------------------
P3085_StatePB.AutoPB := System.Cnvyr_Auto;
P3085_StatePB.ManPB := System.Cnvyr_Manual;
P3085_StatePB.ResetPB := System.Cnvyr_Reset;
P3085_StatePB.OfflinePB := System.Cnvyr_Offline;
P3085SleepWakeTrig[1] := Photoeyes.PE_9191.out;
P3085SleepWakeTrig[2] := GVL_IO.PB_RemoteReset_8251;


// Initialize the Equipment Type
P3085_Status.Sts_EquipmentState.EquipType := E_EquipType.Conveyor;

// Interlocks
//P3085.In_EquipIntlks.2:= 
//Events
P3085.In_EquipEvents.2:= GVL_IO.DS_P3085;
P3085.In_EquipEvents.3:= System.SysEventsAllOk;
P3085.In_EquipEvents.4:= NOT CommStatus.RIO12182_CommFault.Out;
P3085.In_EquipEvents.5:= NOT GVL_IO.P3085_Faulted;

// Function Call
P3085(
   In_p_EquipStatePB:= P3085_StatePB,
   In_P_ConvReqRun:= TRUE,
   In_ConvDwnStrmMtrStatus:=  P3090_Status.Sts_IsRunning,
   In_ConvCrntExitPhotoEye:= Photoeyes.PE_12091.Out,
   In_SimActive:= System.Sys_SimActive,
   In_EquipInit:= GVL_IO.INIT,
   In_WakeSlpTrigArry:= P3085SleepWakeTrig,
   Cfg_EquipIndex := GVL_EquipArrays.nEquipIndex,
   Cfg_EquipLabel := cfgP3085Label,
   Cfg_EquipDefState:= System.ConvDefaultState,
   Cfg_EquipIntlksArry:= cfgP3085IntlksArry,
   Cfg_EquipEvntsArry:= cfgP3085EvntsArry,
   cfg_JamDetectTime:= cfgP3085JamDetectTime,
   Cfg_UseSleepTmr := TRUE,
   Cfg_UseStartUpDelay := TRUE,
   Cfg_StartUpDelayTime := T#500MS,
   Cfg_SleepWaitTime:= cfgP3085SleepTime,
   Sts_EquipState := P3085_Status,
   Out_ConvCrntMtr => GVL_IO.P3085_RUN);

P3085_Status.Sts_IsRunning := GVL_IO.P3085_RUN;
//Transport
//----------------------------------------P3090--------------------------------------------------------------
P3090_StatePB.AutoPB := System.Cnvyr_Auto;
P3090_StatePB.ManPB := System.Cnvyr_Manual;
P3090_StatePB.ResetPB := System.Cnvyr_Reset;
P3090_StatePB.OfflinePB := System.Cnvyr_Offline;
P3090SleepWakeTrig[1] := Photoeyes.PE_12091.out;
P3090SleepWakeTrig[2] := Photoeyes.PE_9191.out;
P3090SleepWakeTrig[3] := GVL_IO.PB_RemoteReset_8251;

// Initialize the Equipment Type
P3090_Status.Sts_EquipmentState.EquipType := E_EquipType.Conveyor;

// Interlocks
//P3090.In_EquipIntlks.2:=
//Events
P3090.In_EquipEvents.2:= GVL_IO.DS_P3090;
P3090.In_EquipEvents.3:= System.SysEventsAllOk;
P3090.In_EquipEvents.4:= NOT CommStatus.RIO12182_CommFault.Out;
P3090.In_EquipEvents.5:= NOT GVL_IO.P3090_Faulted;

// Function Call
P3090(
   In_p_EquipStatePB:= P3090_StatePB,
   In_P_ConvReqRun:= TRUE,
   In_ConvDwnStrmMtrStatus:= P3095_Status.Sts_IsRunning,
   In_ConvCrntExitPhotoEye:=  Photoeyes.PE_12271.out,
   In_SimActive:= System.Sys_SimActive,
   In_EquipInit:= GVL_IO.INIT,
   In_WakeSlpTrigArry:= P3090SleepWakeTrig,
   Cfg_EquipIndex := GVL_EquipArrays.nEquipIndex,
   Cfg_EquipLabel := cfgP3090Label,
   Cfg_EquipDefState:= System.ConvDefaultState,
   Cfg_EquipIntlksArry:= cfgP3090IntlksArry,
   Cfg_EquipEvntsArry:= cfgP3090EvntsArry,
   cfg_JamDetectTime:= cfgP3090JamDetectTime,
   Cfg_UseSleepTmr := TRUE,
   Cfg_UseStartUpDelay := FALSE,
   Cfg_SleepWaitTime:= cfgP3090SleepTime,
   Sts_EquipState := P3090_Status,
   Out_ConvCrntMtr => GVL_IO.P3090_RUN);

P3090_Status.Sts_IsRunning := GVL_IO.P3090_RUN;
//Transport
//----------------------------------------P3095--------------------------------------------------------------
P3095_StatePB.AutoPB := System.Cnvyr_Auto;
P3095_StatePB.ManPB := System.Cnvyr_Manual;
P3095_StatePB.ResetPB := System.Cnvyr_Reset;
P3095_StatePB.OfflinePB := System.Cnvyr_Offline;
P3095SleepWakeTrig[1] := Photoeyes.PE_12271.out OR Photoeyes.PE_9191.out;;
P3095SleepWakeTrig[2] := Photoeyes.PE_12091.out;
P3095SleepWakeTrig[3] := GVL_IO.PB_RemoteReset_8251;

// Initialize the Equipment Type
P3095_Status.Sts_EquipmentState.EquipType := E_EquipType.Conveyor;

// Interlocks
//P3095.In_EquipIntlks.2:= 
//Events
P3095.In_EquipEvents.2:= GVL_IO.DS_P3095;
P3095.In_EquipEvents.3:= System.SysEventsAllOk;
P3095.In_EquipEvents.4:= NOT CommStatus.RIO12182_CommFault.Out;
P3095.In_EquipEvents.5:= ProxSensors.PX_12251_Extended.Out;
P3095.In_EquipEvents.6:= NOT GVL_IO.P3095_Faulted;

// Function Call
P3095(
   In_p_EquipStatePB:= P3095_StatePB,
   In_P_ConvReqRun:= TRUE,
   In_ConvDwnStrmMtrStatus:= GVL_IO.From205_P3100_IsRunning, //EAP Status
   In_ConvCrntExitPhotoEye:= Photoeyes.PE_12181.Out,
   In_SimActive:= System.Sys_SimActive,
   In_EquipInit:= GVL_IO.INIT,
   In_WakeSlpTrigArry:= P3095SleepWakeTrig,
   Cfg_EquipIndex := GVL_EquipArrays.nEquipIndex,
   Cfg_EquipLabel := cfgP3095Label,
   Cfg_EquipDefState:= System.ConvDefaultState,
   Cfg_EquipIntlksArry:= cfgP3095IntlksArry,
   Cfg_EquipEvntsArry:= cfgP3095EvntsArry,
   cfg_JamDetectTime:= cfgP3095JamDetectTime,
   Cfg_UseSleepTmr := TRUE,
   Cfg_SleepWaitTime:= cfgP3095SleepTime,
   Sts_EquipState := P3095_Status,
   Out_ConvCrntMtr => GVL_IO.P3095_RUN);

P3095_Status.Sts_IsRunning := GVL_IO.P3095_RUN;

//Conveyors Incoming 2000 (Purple line)
//Transport
//P2130
//    Remote Index Check
IF Conveyors.P2130_Status.Sts_EquipmentState.Index > 0 THEN
  IF GVL_EquipArrays.aEquipStatusArray_Out[Conveyors.P2130_Status.Sts_EquipmentState.Index].RemIndex <> 0 THEN
      IF Conveyors.P2130_Status.Sts_EquipmentState.RemIndex = 0 THEN
          Conveyors.P2130_Status.Sts_EquipmentState.RemIndex := GVL_EquipArrays.aEquipStatusArray_Out[Conveyors.P2130_Status.Sts_EquipmentState.Index].RemIndex;
      END_IF
  END_IF
  //    Last Operational State Check
  IF GVL_EquipArrays.aEquipStatusArray_Out[Conveyors.P2130_Status.Sts_EquipmentState.Index].LstOperState <> Conveyors.P2130_Status.Sts_EquipmentState.LstOperState THEN
      Conveyors.P2130_Status.Sts_EquipmentState.LstOperState := GVL_EquipArrays.aEquipStatusArray_In[Conveyors.P2130_Status.Sts_EquipmentState.Index].LstOperState;
  END_IF
  //Prepare the Equipment Status data item
  GVL_EquipArrays.aEquipStatusArray_In[Conveyors.P2130_Status.Sts_EquipmentState.Index] := Conveyors.P2130_Status.Sts_EquipmentState;
END_IF
//Transport
//P2135
//    Remote Index Check
IF Conveyors.P2135_Status.Sts_EquipmentState.Index > 0 THEN
  IF GVL_EquipArrays.aEquipStatusArray_Out[Conveyors.P2135_Status.Sts_EquipmentState.Index].RemIndex <> 0 THEN
      IF Conveyors.P2135_Status.Sts_EquipmentState.RemIndex = 0 THEN
          Conveyors.P2135_Status.Sts_EquipmentState.RemIndex := GVL_EquipArrays.aEquipStatusArray_Out[Conveyors.P2135_Status.Sts_EquipmentState.Index].RemIndex;
      END_IF
  END_IF
  //    Last Operational State Check
  IF GVL_EquipArrays.aEquipStatusArray_Out[Conveyors.P2135_Status.Sts_EquipmentState.Index].LstOperState <> Conveyors.P2135_Status.Sts_EquipmentState.LstOperState THEN
      Conveyors.P2135_Status.Sts_EquipmentState.LstOperState := GVL_EquipArrays.aEquipStatusArray_In[Conveyors.P2135_Status.Sts_EquipmentState.Index].LstOperState;
  END_IF
  //Prepare the Equipment Status data item
  GVL_EquipArrays.aEquipStatusArray_In[Conveyors.P2135_Status.Sts_EquipmentState.Index] := Conveyors.P2135_Status.Sts_EquipmentState;
END_IF
//Transport
//P2140
//    Remote Index Check
IF Conveyors.P2140_Status.Sts_EquipmentState.Index > 0 THEN
  IF GVL_EquipArrays.aEquipStatusArray_Out[Conveyors.P2140_Status.Sts_EquipmentState.Index].RemIndex <> 0 THEN
      IF Conveyors.P2140_Status.Sts_EquipmentState.RemIndex = 0 THEN
          Conveyors.P2140_Status.Sts_EquipmentState.RemIndex := GVL_EquipArrays.aEquipStatusArray_Out[Conveyors.P2140_Status.Sts_EquipmentState.Index].RemIndex;
      END_IF
  END_IF
  //    Last Operational State Check
  IF GVL_EquipArrays.aEquipStatusArray_Out[Conveyors.P2140_Status.Sts_EquipmentState.Index].LstOperState <> Conveyors.P2140_Status.Sts_EquipmentState.LstOperState THEN
      Conveyors.P2140_Status.Sts_EquipmentState.LstOperState := GVL_EquipArrays.aEquipStatusArray_In[Conveyors.P2140_Status.Sts_EquipmentState.Index].LstOperState;
  END_IF
  //Prepare the Equipment Status data item
  GVL_EquipArrays.aEquipStatusArray_In[Conveyors.P2140_Status.Sts_EquipmentState.Index] := Conveyors.P2140_Status.Sts_EquipmentState;
END_IF
//Transport
//P2143
//    Remote Index Check
IF Conveyors.P2143_Status.Sts_EquipmentState.Index > 0 THEN
  IF GVL_EquipArrays.aEquipStatusArray_Out[Conveyors.P2143_Status.Sts_EquipmentState.Index].RemIndex <> 0 THEN
      IF Conveyors.P2143_Status.Sts_EquipmentState.RemIndex = 0 THEN
          Conveyors.P2143_Status.Sts_EquipmentState.RemIndex := GVL_EquipArrays.aEquipStatusArray_Out[Conveyors.P2143_Status.Sts_EquipmentState.Index].RemIndex;
      END_IF
  END_IF
  //    Last Operational State Check
  IF GVL_EquipArrays.aEquipStatusArray_Out[Conveyors.P2143_Status.Sts_EquipmentState.Index].LstOperState <> Conveyors.P2143_Status.Sts_EquipmentState.LstOperState THEN
      Conveyors.P2143_Status.Sts_EquipmentState.LstOperState := GVL_EquipArrays.aEquipStatusArray_In[Conveyors.P2143_Status.Sts_EquipmentState.Index].LstOperState;
  END_IF
  //Prepare the Equipment Status data item
  GVL_EquipArrays.aEquipStatusArray_In[Conveyors.P2143_Status.Sts_EquipmentState.Index] := Conveyors.P2143_Status.Sts_EquipmentState;
END_IF
//Spiral
//P2141
//    Remote Index Check
IF Conveyors.P2141_Status.Sts_EquipmentState.Index > 0 THEN
  IF GVL_EquipArrays.aEquipStatusArray_Out[Conveyors.P2141_Status.Sts_EquipmentState.Index].RemIndex <> 0 THEN
      IF Conveyors.P2141_Status.Sts_EquipmentState.RemIndex = 0 THEN
          Conveyors.P2141_Status.Sts_EquipmentState.RemIndex := GVL_EquipArrays.aEquipStatusArray_Out[Conveyors.P2141_Status.Sts_EquipmentState.Index].RemIndex;
      END_IF
  END_IF
  //    Last Operational State Check
  IF GVL_EquipArrays.aEquipStatusArray_Out[Conveyors.P2141_Status.Sts_EquipmentState.Index].LstOperState <> Conveyors.P2141_Status.Sts_EquipmentState.LstOperState THEN
      Conveyors.P2141_Status.Sts_EquipmentState.LstOperState := GVL_EquipArrays.aEquipStatusArray_In[Conveyors.P2141_Status.Sts_EquipmentState.Index].LstOperState;
  END_IF
  //Prepare the Equipment Status data item
  GVL_EquipArrays.aEquipStatusArray_In[Conveyors.P2141_Status.Sts_EquipmentState.Index] := Conveyors.P2141_Status.Sts_EquipmentState;
END_IF
//Transport
//P2142
//    Remote Index Check
IF Conveyors.P2142_Status.Sts_EquipmentState.Index > 0 THEN
  IF GVL_EquipArrays.aEquipStatusArray_Out[Conveyors.P2142_Status.Sts_EquipmentState.Index].RemIndex <> 0 THEN
      IF Conveyors.P2142_Status.Sts_EquipmentState.RemIndex = 0 THEN
          Conveyors.P2142_Status.Sts_EquipmentState.RemIndex := GVL_EquipArrays.aEquipStatusArray_Out[Conveyors.P2142_Status.Sts_EquipmentState.Index].RemIndex;
      END_IF
  END_IF
  //    Last Operational State Check
  IF GVL_EquipArrays.aEquipStatusArray_Out[Conveyors.P2142_Status.Sts_EquipmentState.Index].LstOperState <> Conveyors.P2142_Status.Sts_EquipmentState.LstOperState THEN
      Conveyors.P2142_Status.Sts_EquipmentState.LstOperState := GVL_EquipArrays.aEquipStatusArray_In[Conveyors.P2142_Status.Sts_EquipmentState.Index].LstOperState;
  END_IF
  //Prepare the Equipment Status data item
  GVL_EquipArrays.aEquipStatusArray_In[Conveyors.P2142_Status.Sts_EquipmentState.Index] := Conveyors.P2142_Status.Sts_EquipmentState;
END_IF
//Transport
//P2145
//    Remote Index Check
IF Conveyors.P2145_Status.Sts_EquipmentState.Index > 0 THEN
  IF GVL_EquipArrays.aEquipStatusArray_Out[Conveyors.P2145_Status.Sts_EquipmentState.Index].RemIndex <> 0 THEN
      IF Conveyors.P2145_Status.Sts_EquipmentState.RemIndex = 0 THEN
          Conveyors.P2145_Status.Sts_EquipmentState.RemIndex := GVL_EquipArrays.aEquipStatusArray_Out[Conveyors.P2145_Status.Sts_EquipmentState.Index].RemIndex;
      END_IF
  END_IF
  //    Last Operational State Check
  IF GVL_EquipArrays.aEquipStatusArray_Out[Conveyors.P2145_Status.Sts_EquipmentState.Index].LstOperState <> Conveyors.P2145_Status.Sts_EquipmentState.LstOperState THEN
      Conveyors.P2145_Status.Sts_EquipmentState.LstOperState := GVL_EquipArrays.aEquipStatusArray_In[Conveyors.P2145_Status.Sts_EquipmentState.Index].LstOperState;
  END_IF
  //Prepare the Equipment Status data item
  GVL_EquipArrays.aEquipStatusArray_In[Conveyors.P2145_Status.Sts_EquipmentState.Index] := Conveyors.P2145_Status.Sts_EquipmentState;
END_IF
//Spiral
//P2146
//    Remote Index Check
IF Conveyors.P2146_Status.Sts_EquipmentState.Index > 0 THEN
  IF GVL_EquipArrays.aEquipStatusArray_Out[Conveyors.P2146_Status.Sts_EquipmentState.Index].RemIndex <> 0 THEN
      IF Conveyors.P2146_Status.Sts_EquipmentState.RemIndex = 0 THEN
          Conveyors.P2146_Status.Sts_EquipmentState.RemIndex := GVL_EquipArrays.aEquipStatusArray_Out[Conveyors.P2146_Status.Sts_EquipmentState.Index].RemIndex;
      END_IF
  END_IF
  //    Last Operational State Check
  IF GVL_EquipArrays.aEquipStatusArray_Out[Conveyors.P2146_Status.Sts_EquipmentState.Index].LstOperState <> Conveyors.P2146_Status.Sts_EquipmentState.LstOperState THEN
      Conveyors.P2146_Status.Sts_EquipmentState.LstOperState := GVL_EquipArrays.aEquipStatusArray_In[Conveyors.P2146_Status.Sts_EquipmentState.Index].LstOperState;
  END_IF
  //Prepare the Equipment Status data item
  GVL_EquipArrays.aEquipStatusArray_In[Conveyors.P2146_Status.Sts_EquipmentState.Index] := Conveyors.P2146_Status.Sts_EquipmentState;
END_IF
//Sorter
//P2150
//    Remote Index Check
IF Conveyors.P2150_Status.Sts_EquipmentState.Index > 0 THEN
  IF GVL_EquipArrays.aEquipStatusArray_Out[Conveyors.P2150_Status.Sts_EquipmentState.Index].RemIndex <> 0 THEN
      IF Conveyors.P2150_Status.Sts_EquipmentState.RemIndex = 0 THEN
          Conveyors.P2150_Status.Sts_EquipmentState.RemIndex := GVL_EquipArrays.aEquipStatusArray_Out[Conveyors.P2150_Status.Sts_EquipmentState.Index].RemIndex;
      END_IF
  END_IF
  //    Last Operational State Check
  IF GVL_EquipArrays.aEquipStatusArray_Out[Conveyors.P2150_Status.Sts_EquipmentState.Index].LstOperState <> Conveyors.P2150_Status.Sts_EquipmentState.LstOperState THEN
      Conveyors.P2150_Status.Sts_EquipmentState.LstOperState := GVL_EquipArrays.aEquipStatusArray_In[Conveyors.P2150_Status.Sts_EquipmentState.Index].LstOperState;
  END_IF
  //Prepare the Equipment Status data item
  GVL_EquipArrays.aEquipStatusArray_In[Conveyors.P2150_Status.Sts_EquipmentState.Index] := Conveyors.P2150_Status.Sts_EquipmentState;
END_IF
//Conveyors Incoming 3000 (Green line)
//Spiral
//P3080
//    Remote Index Check
IF Conveyors.P3080_Status.Sts_EquipmentState.Index > 0 THEN
  IF GVL_EquipArrays.aEquipStatusArray_Out[Conveyors.P3080_Status.Sts_EquipmentState.Index].RemIndex <> 0 THEN
      IF Conveyors.P3080_Status.Sts_EquipmentState.RemIndex = 0 THEN
          Conveyors.P3080_Status.Sts_EquipmentState.RemIndex := GVL_EquipArrays.aEquipStatusArray_Out[Conveyors.P3080_Status.Sts_EquipmentState.Index].RemIndex;
      END_IF
  END_IF
  //    Last Operational State Check
  IF GVL_EquipArrays.aEquipStatusArray_Out[Conveyors.P3080_Status.Sts_EquipmentState.Index].LstOperState <> Conveyors.P3080_Status.Sts_EquipmentState.LstOperState THEN
      Conveyors.P3080_Status.Sts_EquipmentState.LstOperState := GVL_EquipArrays.aEquipStatusArray_In[Conveyors.P3080_Status.Sts_EquipmentState.Index].LstOperState;
  END_IF
  //Prepare the Equipment Status data item
  GVL_EquipArrays.aEquipStatusArray_In[Conveyors.P3080_Status.Sts_EquipmentState.Index] := Conveyors.P3080_Status.Sts_EquipmentState;
END_IF
//Transport
//P3085
//    Remote Index Check
IF Conveyors.P3085_Status.Sts_EquipmentState.Index > 0 THEN
  IF GVL_EquipArrays.aEquipStatusArray_Out[Conveyors.P3085_Status.Sts_EquipmentState.Index].RemIndex <> 0 THEN
      IF Conveyors.P3085_Status.Sts_EquipmentState.RemIndex = 0 THEN
          Conveyors.P3085_Status.Sts_EquipmentState.RemIndex := GVL_EquipArrays.aEquipStatusArray_Out[Conveyors.P3085_Status.Sts_EquipmentState.Index].RemIndex;
      END_IF
  END_IF
  //    Last Operational State Check
  IF GVL_EquipArrays.aEquipStatusArray_Out[Conveyors.P3085_Status.Sts_EquipmentState.Index].LstOperState <> Conveyors.P3085_Status.Sts_EquipmentState.LstOperState THEN
      Conveyors.P3085_Status.Sts_EquipmentState.LstOperState := GVL_EquipArrays.aEquipStatusArray_In[Conveyors.P3085_Status.Sts_EquipmentState.Index].LstOperState;
  END_IF
  //Prepare the Equipment Status data item
  GVL_EquipArrays.aEquipStatusArray_In[Conveyors.P3085_Status.Sts_EquipmentState.Index] := Conveyors.P3085_Status.Sts_EquipmentState;
END_IF
//Transport
//P3090
//    Remote Index Check
IF Conveyors.P3090_Status.Sts_EquipmentState.Index > 0 THEN
  IF GVL_EquipArrays.aEquipStatusArray_Out[Conveyors.P3090_Status.Sts_EquipmentState.Index].RemIndex <> 0 THEN
      IF Conveyors.P3090_Status.Sts_EquipmentState.RemIndex = 0 THEN
          Conveyors.P3090_Status.Sts_EquipmentState.RemIndex := GVL_EquipArrays.aEquipStatusArray_Out[Conveyors.P3090_Status.Sts_EquipmentState.Index].RemIndex;
      END_IF
  END_IF
  //    Last Operational State Check
  IF GVL_EquipArrays.aEquipStatusArray_Out[Conveyors.P3090_Status.Sts_EquipmentState.Index].LstOperState <> Conveyors.P3090_Status.Sts_EquipmentState.LstOperState THEN
      Conveyors.P3090_Status.Sts_EquipmentState.LstOperState := GVL_EquipArrays.aEquipStatusArray_In[Conveyors.P3090_Status.Sts_EquipmentState.Index].LstOperState;
  END_IF
  //Prepare the Equipment Status data item
  GVL_EquipArrays.aEquipStatusArray_In[Conveyors.P3090_Status.Sts_EquipmentState.Index] := Conveyors.P3090_Status.Sts_EquipmentState;
END_IF
//Transport
//P3095
//    Remote Index Check
IF Conveyors.P3095_Status.Sts_EquipmentState.Index > 0 THEN
  IF GVL_EquipArrays.aEquipStatusArray_Out[Conveyors.P3095_Status.Sts_EquipmentState.Index].RemIndex <> 0 THEN
      IF Conveyors.P3095_Status.Sts_EquipmentState.RemIndex = 0 THEN
          Conveyors.P3095_Status.Sts_EquipmentState.RemIndex := GVL_EquipArrays.aEquipStatusArray_Out[Conveyors.P3095_Status.Sts_EquipmentState.Index].RemIndex;
      END_IF
  END_IF
  //    Last Operational State Check
  IF GVL_EquipArrays.aEquipStatusArray_Out[Conveyors.P3095_Status.Sts_EquipmentState.Index].LstOperState <> Conveyors.P3095_Status.Sts_EquipmentState.LstOperState THEN
      Conveyors.P3095_Status.Sts_EquipmentState.LstOperState := GVL_EquipArrays.aEquipStatusArray_In[Conveyors.P3095_Status.Sts_EquipmentState.Index].LstOperState;
  END_IF
  //Prepare the Equipment Status data item
  GVL_EquipArrays.aEquipStatusArray_In[Conveyors.P3095_Status.Sts_EquipmentState.Index] := Conveyors.P3095_Status.Sts_EquipmentState;
END_IF

END_PROGRAM

// ---- FunctionBlocks/Conveyance/FB_CnvyrCnfig_1.TcPOU
FUNCTION_BLOCK FB_CnvyrCnfig_1

(* Standard Conveyor Set up,
	Uses Interlocks. Has 14 that can be assigned that are conveyor specific and a common interlock for exit conveyor PE and Dwn Stream MTR status
	Has an interlock for System.SysIntlksAllOk
	Doesn't use Start Conditions  
	Uses Events and has 15 that can be assigned that are conveyor specific and a common event for the exit conveyor PE Jam detected fault  *)
(* End Conveyor Set up,
	This configuration doesn't use the downstream motor status
	Uses Interlocks. Has 14 that can be assigned that are conveyor specific and a common interlock for conveyor full using the exit PE of this conveyor
	Has an interlock for System.SysIntlksAllOk
	Doesn't use Start Conditions  
	Uses Events and has 16 that can be assigned that are conveyor specific *)
(* Slave Conveyor Set up,
	Uses Interlocks. Has 14 that can be assigned that are conveyor specific and a common interlock for Dwn Stream MTR status
	Has an interlock for System.SysIntlksAllOk
	Doesn't use Start Conditions  
	Uses Events and has 16 that can be assigned that are conveyor specifi  *)

VAR_IN_OUT
	CFG_EquipIndex				: DINT;	// Index used for local Equipment status array
	{attribute 'OPC.UA.DA' := '1'}
	Sts_EquipState				: ST_EquipmentStatus;		// State Status
//	In_EquipEvents				: UINT;		// Events that are specific to the instance of the conveyor
//	In_EquipIntlks				: UINT;		// Interlock that is specific to the instance of the conveyor
END_VAR
VAR_INPUT
	{attribute 'OPC.UA.DA' := '1'}
	In_o_EquipStatePB			: ST_StateCntrlPB;		// Hmi push butons to change states
	In_p_EquipStatePB			: ST_StateCntrlPB;		// programming to change states
	In_P_ConvReqRun				: BOOL;		// Input to start output if in auto and conditions are met
	In_ConvDwnStrmMtrStatus		: BOOL;		// The Down Stearm Motors Status (0= OFF, 1= ON/Running)
	In_ConvCrntExitPhotoEye		: BOOL;		// The Current Photo Eye (1= blocked)
	In_SimActive				: BOOL;
	In_EquipInit					: BOOL;		// Initialise;
	In_EquipMtrFdbck			: BOOL := FALSE;	// Motor Running Feedback (1 = Running), VFD or Contactor
	Cfg_EquipDefState			: E_StateCntrl;
	{attribute 'OPC.UA.DA' := '1'}
	Cfg_EquipLabel				: STRING(20);		// Label of the conveyor
	Cfg_UseMtrFdbck				: BOOL := FALSE;	// Use Feedback from Contactor or VFD 
	Cfg_UseStartUpDelay			: BOOL := FALSE;	// Use a Start-up Delay
	Cfg_StartUpDelayTime		: TIME := T#1S;		// Start-up delay time
	Cfg_InvertMotorOut          : BOOL := FALSE;
	Cfg_ConvType				: E_ConvType := E_ConvType.standard;	// Default to a standard conveyor type
	Cfg_JamDetectTime			: TIME;
	
	// Events
	{attribute 'OPC.UA.DA' := '0'}
	Cfg_EquipEvntsArry			: ARRAY [0..15] OF ST_CfgEvents;
	In_EquipEvents				: UINT;		// Events that are specific to the instance of the conveyor
	
	// Interlocks that can be Instance Specific
	{attribute 'OPC.UA.DA' := '0'}
	Cfg_EquipIntlksArry			: ARRAY [0..15] OF ST_CfgEvents;		// Descriptions of the Interlock 
	In_EquipIntlks				: UINT;		// Interlock that is specific to the instance of the conveyor
	// Sleep Timer	
	Cfg_UseSleepTmr				: BOOL;	// Configure sleep or not sleep this conveyor
	In_WakeSlpTrigArry			: ARRAY [1..5] OF BOOL;		// Input to watch (or wake) for sleep timer
	Cfg_SleepWaitTime			: TIME;		// Time to Wait after last Input before sleeping
	
END_VAR
VAR_OUTPUT
	{attribute 'OPC.UA.DA' := '1'}
	Out_ConvCrntMtr				: BOOL;		// Run command for the current motor
	{attribute 'OPC.UA.DA' := '1'}
	Out_ConvCrntMtr_Raw			: BOOL;		// Run command for the current motor
	{attribute 'OPC.UA.DA' := '1'}
	Sts_ConvCrntMtr				: BOOL;		// Status showing that current motor is running
	{attribute 'OPC.UA.DA' := '1'}
	Sts_ConvSleepingActive		: BOOL;
	{attribute 'OPC.UA.DA' := '1'}
	Sts_All_Intlks_OK			: BOOL;		// Status bit to show that all interloks are good to Run 
	{attribute 'OPC.UA.DA' := '1'}
	Sts_FaultActive				: BOOL;	// Status Bit Showing that a fault is present (0= No Active Faults, 1= Fault Active)
	{attribute 'OPC.UA.DA' := '1'}
	Sts_WarnActive				: BOOL;	// Status Bit Showing that a warning is present (0= No Active Warnings, 1= Warning Active)
	{attribute 'OPC.UA.DA' := '1'}
	Sts_All_Evnts_OK			: BOOL;		// Status Bit Showing that ALL Events are OK to RUN (0= Event Present, 1= OK to Run)
	{attribute 'OPC.UA.DA' := '1'}
	Sts_IntlksArry				: ARRAY[0..15] OF ST_EventSts;		// Interlock status 0 to 15 Input
	{attribute 'OPC.UA.DA' := '1'}
	Sts_FaultsArry				: ARRAY[0..15] OF ST_EventSts;	// Status of each Fault Event State (0= OFF, 1=ON)
	{attribute 'OPC.UA.DA' := '1'}
	Sts_WarnsArry				: ARRAY[0..15] OF ST_EventSts;		// Status of each Warning Event State (0= OFF, 1=ON)
	{attribute 'OPC.UA.DA' := '0'}
	Sts_EvntsArry				: ARRAY[0..15] OF ST_EventSts; 	// Status of each Event State (0= OFF, 1=ON)
END_VAR
VAR
	{attribute 'OPC.UA.DA' := '0'}
	Conv_fbIntrlks				: FB_Intlks_Latch;
	Conv_IntlksArry				: ARRAY[0..15] OF BOOL;
	{attribute 'OPC.UA.DA' := '0'}
	Conv_fbEquipCntrl			: FB_EquipCntrl;
	{attribute 'OPC.UA.DA' := '0'}
	Conv_EventManager			: FB_EventMngr;
	Conv_CrrntExitPEJamDetctd	: FB_JamDetect;
	Conv_EventArry				: ARRAY[0..15] OF BOOL;
	
	Conv_LatchIgnore			: BOOL := FALSE;		// Put as a place holder for ease of future use
	Conv_LatchReset				: BOOL := FALSE;		//Put as a place holder for ease of future use
	Conv_IntlkBypassed			: ARRAY [0..15] OF BOOL;		//Put as a place holder for ease of future use
	Conv_RunEnabled				: BOOL;					// TRUE = Enable the conveyor to run
	Conv_StartEnabled			: BOOL;					// TRUE = Start Motion for Conv Enabled
	Conv_StartAllowed			: BOOL;					// TRUE = Start Motion for Conv Allowed

	// Sleep Timer
	fbSleepCntrl				: FB_SleepCntrl;

	// Start-up Delay Timer
	tStartUpDelay				: TON;

END_VAR

(*
	Depending on the conveyor type, the Interlock and Event 0 is different
	Also, jams are only detected on standard and end conveyors

	If no valid conveyor type is specified, the default is a standard type
*)

CASE Cfg_ConvType OF
	E_ConvType.standard:
		Conv_IntlksArry[0] := In_ConvDwnStrmMtrStatus OR (NOT In_ConvDwnStrmMtrStatus AND NOT In_ConvCrntExitPhotoEye);
		Conv_EventArry[0] := Conv_CrrntExitPEJamDetctd.JamDetected;
		Conv_CrrntExitPEJamDetctd(
			In_PE:= In_ConvCrntExitPhotoEye 
					AND NOT Sts_EquipState.Sts_EquipmentState.StsOffline 
					AND NOT In_o_EquipStatePB.ResetPB 
					AND NOT In_p_EquipStatePB.ResetPB, 
			In_Status:= Out_ConvCrntMtr_Raw, 
			CFG_PEOKState:= 0, 
			JamDetTime:= cfg_JamDetectTime);
	E_ConvType.end:
		Conv_IntlksArry[0] := Conv_CrrntExitPEJamDetctd.JamDetected;
		Conv_EventArry[0] := In_EquipEvents.0;
		Conv_CrrntExitPEJamDetctd(
			In_PE:= In_ConvCrntExitPhotoEye 
					AND NOT Sts_EquipState.Sts_EquipmentState.StsOffline 
					AND NOT In_o_EquipStatePB.ResetPB 
					AND NOT In_p_EquipStatePB.ResetPB, 
			In_Status:= Out_ConvCrntMtr_Raw, 
			CFG_PEOKState:= 0, 
			JamDetTime:= cfg_JamDetectTime);
	E_ConvType.slave:
		Conv_IntlksArry[0] := In_ConvDwnStrmMtrStatus;
		Conv_EventArry[0] := In_EquipEvents.0;
	ELSE
		Conv_IntlksArry[0] := In_ConvDwnStrmMtrStatus OR (NOT In_ConvDwnStrmMtrStatus AND NOT In_ConvCrntExitPhotoEye);
		Conv_EventArry[0] := Conv_CrrntExitPEJamDetctd.JamDetected;
		Conv_CrrntExitPEJamDetctd(
			In_PE:= In_ConvCrntExitPhotoEye 
					AND NOT Sts_EquipState.Sts_EquipmentState.StsOffline 
					AND NOT In_o_EquipStatePB.ResetPB 
					AND NOT In_p_EquipStatePB.ResetPB, 
			In_Status:= Out_ConvCrntMtr_Raw, 
			CFG_PEOKState:= 0, 
			JamDetTime:= cfg_JamDetectTime);
END_CASE
// Set Up Common Converyor Interlocks and inputs for interlocks
Conv_IntlksArry[1] := System.SysIntlksAllOk; 
Conv_IntlksArry[2] := In_EquipIntlks.2;
Conv_IntlksArry[3] := In_EquipIntlks.3;
Conv_IntlksArry[4] := In_EquipIntlks.4;
Conv_IntlksArry[5] := In_EquipIntlks.5;
Conv_IntlksArry[6] := In_EquipIntlks.6;
Conv_IntlksArry[7] := In_EquipIntlks.7;
Conv_IntlksArry[8] := In_EquipIntlks.8;
Conv_IntlksArry[9] := In_EquipIntlks.9; 
Conv_IntlksArry[10] := In_EquipIntlks.10;
Conv_IntlksArry[11] := In_EquipIntlks.11;
Conv_IntlksArry[12] := In_EquipIntlks.12;
Conv_IntlksArry[13] := In_EquipIntlks.13;
Conv_IntlksArry[14] := In_EquipIntlks.14;
Conv_IntlksArry[15] := Conv_StartAllowed;
	


// Call Interlock block
Conv_fbIntrlks(
	In_Intlks:= Conv_IntlksArry,
	CFG_IntlksArry:= Cfg_EquipIntlksArry, 
	HMI_LatchIgnore:= Conv_LatchIgnore, 
	HMI_LatchReset:= Conv_LatchReset, 
	All_Intlk_OK=> Sts_EquipState.Sts_All_Intlks_OK, 
	STS_Intlks=> Sts_IntlksArry);
	
// Set Up Common Converyor Events and inputs for events
Conv_EventArry[1]:=	In_EquipEvents.1;
Conv_EventArry[2]:= In_EquipEvents.2;
Conv_EventArry[3]:= In_EquipEvents.3;
Conv_EventArry[4]:= In_EquipEvents.4;
Conv_EventArry[5]:= In_EquipEvents.5;
Conv_EventArry[6]:= In_EquipEvents.6;
Conv_EventArry[7]:= In_EquipEvents.7;
Conv_EventArry[8]:= In_EquipEvents.8;
Conv_EventArry[9]:= In_EquipEvents.9;
Conv_EventArry[10]:= In_EquipEvents.10;
Conv_EventArry[11]:= In_EquipEvents.11;
Conv_EventArry[12]:= In_EquipEvents.12;
Conv_EventArry[13]:= In_EquipEvents.13;
Conv_EventArry[14]:= In_EquipEvents.14;
Conv_EventArry[15]:= In_EquipEvents.15;

//In_EquipEvents := 0;

// Event Manager
Conv_EventManager(
	sEquipStateCntrlSts := Sts_EquipState.Sts_EquipmentState,
	In_EventsArry := Conv_EventArry ,  
	CFG_EvntsArry:= Cfg_EquipEvntsArry, 
	HMI_LatchReset:= In_o_EquipStatePB.ResetPB OR In_p_EquipStatePB.ResetPB,
	Out_FaultActive=> Sts_EquipState.Sts_FaultActive, 
	Out_WarnActive=> Sts_EquipState.Sts_WarnActive, 
	Sts_All_Evnts_OK=> Sts_EquipState.Sts_All_Evnts_OK, 
	Sts_FaultsArry=> Sts_FaultsArry, 
	Sts_WarnsArry=> Sts_WarnsArry, 
	Sts_EvntsArry=> Sts_EvntsArry);
	
//Call Equipment FB to control current motor	
Conv_fbEquipCntrl(
	CFG_EquipIndex := cfg_EquipIndex,
	CFG_EquipLabel := Cfg_EquipLabel,
	CFG_UseStrtCnd:= FALSE, 
	CFG_UseIntrlks:= TRUE, 
	CFG_UseHrnDly:= Cfg_UseStartUpDelay, 
	CFG_EquipDefState:= Cfg_EquipDefState, 
	In_IntlksOK:= Sts_EquipState.Sts_All_Intlks_OK, 
	In_SimActive:= In_SimActive, 
	In_Init:= In_EquipInit, 
	o_EquipStatePB:= In_o_EquipStatePB, 
	p_EquipStatePB:= In_p_EquipStatePB, 
	P_EquipReqRun:= In_P_ConvReqRun, 
	In_EquipFaults:= Sts_EquipState.Sts_FaultActive, 
	Out_EquipRun=> , 
	Out_Horn=> , 
	Sts_EquipState:= Sts_EquipState.Sts_EquipmentState);	

//===Sleep Timer
IF CFG_UseSleepTmr THEN
	fbSleepCntrl.In_Trigs.0 := In_ConvCrntExitPhotoEye OR In_p_EquipStatePB.AutoPB; 
	fbSleepCntrl.In_Trigs.1 := In_WakeSlpTrigArry[1];
	fbSleepCntrl.In_Trigs.2 := In_WakeSlpTrigArry[2];
	fbSleepCntrl.In_Trigs.3 := In_WakeSlpTrigArry[3];
	fbSleepCntrl.In_Trigs.4 := In_WakeSlpTrigArry[4];
	fbSleepCntrl.In_Trigs.5 := In_WakeSlpTrigArry[5];
	fbSleepCntrl( 
		In_CrntFeedBack:= Out_ConvCrntMtr_Raw, 
		In_ConvState := Sts_EquipState.Sts_EquipmentState.CrntState,
		CFG_WaitToSlpTime:= Cfg_SleepWaitTime,
		SleepActive=> Sts_EquipState.Sts_SleepingActive);
ELSE
	Sts_EquipState.Sts_SleepingActive := FALSE;
END_IF
Sts_ConvSleepingActive := Sts_EquipState.Sts_SleepingActive;

(*
	Process the Conv_StartAllowed signal
	The Conv_StartAllowed enforces the cascade start of conveyors by waiting for the downstream motor to be running before
	this conveyor starts.
	Any conveyor can be started using the Start/Auto push-button without waiting for the downstream conveyor to be running.
*)
IF Sts_EquipState.Sts_EquipmentState.StsAuto THEN
	IF NOT Conv_StartAllowed THEN
		Conv_StartAllowed := In_ConvDwnStrmMtrStatus OR In_o_EquipStatePB.AutoPB OR (Cfg_ConvType = E_ConvType.end) OR (NOT Cfg_UseStartUpDelay);
	END_IF
ELSE
	Conv_StartAllowed := FALSE;
END_IF

// Process the Conv_RunEnabled signal
Conv_RunEnabled := Conv_fbEquipCntrl.Out_EquipRun
				AND NOT (Sts_EquipState.Sts_SleepingActive) 
				AND (Sts_EquipState.Sts_EquipmentState.StsMan OR (Sts_EquipState.Sts_EquipmentState.StsAuto AND Conv_StartAllowed));

// Use or do not use a start-up delay
IF Cfg_UseStartUpDelay THEN
	tStartUpDelay(IN := Conv_RunEnabled
					, PT := Cfg_StartUpDelayTime
					, Q =>);
	IF tStartUpDelay.Q THEN
		Conv_StartEnabled := TRUE;
	ELSE
		Conv_StartEnabled := FALSE;
	END_IF
ELSE
		Conv_StartEnabled := Conv_RunEnabled;	
END_IF

// Run motor based on the results of the Equipment Control and sleeping state
Out_ConvCrntMtr_Raw := Conv_StartEnabled;

// Capture WarnActive to carry these attributes into the Equipment state for System State reporting and display
Sts_EquipState.Sts_EquipmentState.StsHasWarnings := Sts_EquipState.Sts_WarnActive;

// Set Conveyor Motor Running Status
Sts_ConvCrntMtr := (CFG_UseMtrFdbck AND In_EquipMtrFdbck) OR (NOT CFG_UseMtrFdbck AND Out_ConvCrntMtr_Raw) OR (In_SimActive AND Conv_fbEquipCntrl.RunApproved);

// Capture the Operation state of the Conveyor
IF Sts_ConvCrntMtr THEN
	// Conveyor Running
	Sts_EquipState.Sts_EquipmentState.CrntOperState := E_OperStateCntrl.running;
ELSE
	IF Sts_EquipState.Sts_SleepingActive THEN
		// Conveyor Sleeping
		Sts_EquipState.Sts_EquipmentState.CrntOperState := E_OperStateCntrl.sleeping;
	ELSE
		// Conveyor Stopped
		Sts_EquipState.Sts_EquipmentState.CrntOperState := E_OperStateCntrl.stopped;
	END_IF
END_IF

//invert output
IF Cfg_InvertMotorOut THEN
    Out_ConvCrntMtr := NOT Out_ConvCrntMtr_Raw;
ELSE
    Out_ConvCrntMtr := Out_ConvCrntMtr_Raw;
END_IF

// Populate the Sts Output Variables
Sts_All_Intlks_OK  := Sts_EquipState.Sts_All_Intlks_OK;
Sts_All_Evnts_OK  := Sts_EquipState.Sts_All_Evnts_OK;
Sts_FaultActive := Sts_EquipState.Sts_FaultActive;
Sts_WarnActive := Sts_EquipState.Sts_WarnActive;

END_FUNCTION_BLOCK

// ---- FunctionBlocks/Utils/FB_EquipCntrl.TcPOU
(*
=====================================================================
	Copyright ©  Syscon Automation.  All Rights Reserved.
	Version 1 Release 1 2019
	Version 1 Release 2 2020 - Added Initialization for Equipment Label and Index
=====================================================================
 
This FB monitors Start, Interlock and State inputs and controls the output for a motor or other piece of equipment
It is configurable. Choose to use the Start conditions, run interlocks, or horn output
The time the horn sounds and the delay after the horn is sounded are also configurable

*)
FUNCTION_BLOCK FB_EquipCntrl
VAR_IN_OUT
	CFG_EquipIndex		: DINT;	// Index used for local Equipment status array
	Sts_EquipState		: ST_StateCntrlSts;		// State Status
END_VAR
VAR_INPUT
	In_IntlksOK			: BOOL;		// Input for All Interlocks are Good to Run
	In_StartCondsOK		: BOOL;		// Input for All Start Conditions Are Good Run
	In_SimActive		: BOOL;		// Simulation active bit to stop output and send status ignoring feedback (1= Simulation)
	In_ManHrnTrig		: BOOL;		// Manual bit to sound horn for the horn time/duration 
	In_EquipFaults		: BOOL;		// Shutdown Fault input
	In_Init				: BOOL; 

	CFG_UseStrtCnd		: BOOL;		// Bit to use Start conditions (1=use Start conditions)	
	CFG_UseIntrlks		: BOOL;		// Bit to use Interlocks (1=use interlocks)
	CFG_UseHrnDly		: BOOL;		// use horn delay before setting equip/motor output
	CFG_HrnTime			: TIME;		// Time (or duration) for Horn to sound
	CFG_HrnWaitTime		: TIME;		// Time to delay after horn has sounded
	CFG_EquipLabel		: STRING[5];	// Label used to identify the equipment
	CFG_EquipDefState	: E_StateCntrl;	// Default State of Equipment
	
	// State Control
	o_EquipStatePB		: ST_StateCntrlPB;		// Hmi push butons to change states
	p_EquipStatePB		: ST_StateCntrlPB;		// programming to change states
	P_EquipReqRun		: BOOL;		// Input to start output if in auto and conditions are met
		
END_VAR
VAR_OUTPUT
	Out_EquipRun			: BOOL;	// Output for equipment control (1=Run )
	Out_EquipRunInv			: BOOL;	// Inverse of equipment control output
	Out_Horn				: BOOL;	// Output for warning horn or beacon if configured (1=Horn/Beacon ON)
	Sts_EquipIntlksOK		: BOOL;	// Interlock status
	Sts_EquipStartCondOK	: BOOL;	// Start Conditions status 
END_VAR
VAR
	// State Control
	fbStateCntrl			: FB_StateCntrl;

	StartCondPass			: BOOL;
	InterlocksPass			: BOOL;
	RunApproved				: BOOL;
	SoundHornTon			: TON;
	HrnWaitTon				: TON;
	Horn_Rtrig				: R_TRIG;
	Horn_Ftrig				: F_TRIG;
	Horn_Required			: BOOL;
	HornWaitActive			: BOOL;
	HornSoundComplete		: BOOL;
	HornWaitRequired		: BOOL;
	HornDelaysCompleted		: BOOL;
	HornDelaysPass			: BOOL;
	HornOnlyRtrig			: R_TRIG;
	StateStartingRtrig		: R_TRIG;

END_VAR

//===Interlocks
// Check if Conditions are met
InterlocksPass := (In_IntlksOK AND CFG_UseIntrlks AND (Sts_EquipState.StsAuto)) OR (NOT CFG_UseIntrlks) OR (Sts_EquipState.StsMan);

//===State Control
fbStateCntrl(
	CFG_EquipIndex := CFG_EquipIndex,
	CFG_EquipLabel := CFG_EquipLabel,
	o_StatePB:= o_EquipStatePB, 
	p_StatePB:= p_EquipStatePB, 
	P_ReqRun:= P_EquipReqRun, 
	IN_Fault:= In_EquipFaults, 
	IN_Init:= In_Init, 
	CfgDefState:= CFG_EquipDefState, 
	Sts_StateCntrl := Sts_EquipState);
	
// Check for State Start Up Transition
StateStartingRtrig(CLK:=Sts_EquipState.StateRunOK);

//Set eguipment approved to Run
// If it needs to start look at start conditions
IF NOT RunApproved THEN		
	StartCondPass := (In_StartCondsOK AND StateStartingRtrig.Q AND CFG_UseStrtCnd AND (Sts_EquipState.StsAuto)) OR (NOT CFG_UseStrtCnd) OR (Sts_EquipState.StsMan);
	RunApproved := StartCondPass AND InterlocksPass AND Sts_EquipState.StateRunOK;
// If currently running just look at shutdown conditions
ELSE		
	RunApproved := InterlocksPass AND Sts_EquipState.StateRunOK;
END_IF

// Set up rising trigger for horn
Horn_Rtrig(CLK:=(RunApproved AND CFG_UseHrnDly));
IF Horn_Rtrig.Q THEN
	Horn_Required := TRUE;
	HornWaitRequired :=TRUE;
END_IF

HornOnlyRtrig(CLK:=In_ManHrnTrig);
IF HornOnlyRtrig.Q THEN
	Horn_Required := TRUE;
END_IF
	
// Horn timers
SoundHornTon(IN:= Horn_Required , PT:=CFG_HrnTime);
IF SoundHornTon.Q THEN
	Horn_Required:= FALSE;
	IF HornWaitRequired THEN
		HornWaitActive:= TRUE;	
	END_IF	
END_IF

HrnWaitTon(IN:=HornWaitActive, PT:=CFG_HrnWaitTime);
IF HrnWaitTon.Q THEN
	HornWaitActive := FALSE;
	HornWaitRequired := FALSE;
	HornDelaysCompleted := TRUE;	
END_IF

// Set up falling trigger to reset horn bits
Horn_Ftrig(CLK:= RunApproved);
IF Horn_Ftrig.Q THEN
	Horn_Required := FALSE;
	HornWaitRequired := FALSE;
	HornWaitActive:= FALSE;
	HornDelaysCompleted := FALSE;
END_IF

// Set Horn delays
HornDelaysPass := (HornDelaysCompleted AND CFG_UseHrnDly) OR (NOT CFG_UseHrnDly); 

//Set Equipment Output
Out_Horn := Horn_Required;
Out_EquipRun := RunApproved AND HornDelaysPass AND (NOT In_SimActive);
Out_EquipRunInv := NOT Out_EquipRun;

//Set relevant equipment status
Sts_EquipIntlksOK := In_IntlksOK;
Sts_EquipStartCondOK := In_StartCondsOK;

END_FUNCTION_BLOCK

// ---- FunctionBlocks/StateControl/FB_StateCntrl.TcPOU
FUNCTION_BLOCK FB_StateCntrl
(* ==================================================================
	Copyright ©  Syscon Automation.  All Rights Reserved.
	Based on Syscon ConveyorStatus V2 release 1
	Version 1 Release 1 2019
	Version 1 Release 2 2020 - Added Initialization for Equipment Label and Index
	Version 1 Release 3 2020 - Modified for Updated ST_StateCntrlPB and ST_StateCntrlSts structures
=====================================================================
	This function block will control any object’s state based on inputs. 
		The E inputs will change the state anytime they are activated
		The O inputs are conditional based on the current state (eventually these should also be tied to login status) 
		Outputs the current State with troubleshooting status outputs.  
		See Syscon FB Description for more details
---------------------------------------------------------------------
*)
VAR_IN_OUT
	CFG_EquipIndex: 	DINT;				// Index used for local Equipment status array
	Sts_StateCntrl:		ST_StateCntrlSts;	// State Status
END_VAR
VAR_INPUT
	o_StatePB:			ST_StateCntrlPB;	// HMI/manual push buttons to change states
	p_StatePB:			ST_StateCntrlPB;	// programming to change states
	P_ReqRun:			BOOL;				// Input to allow output if in auto and conditions are met
	IN_Fault:			BOOL;				// Fault input
	IN_Init:			BOOL;				// initialization input
	CfgDefState:		E_StateCntrl;
	CFG_EquipLabel:		STRING[5];			// Label used to identify the equipment
END_VAR

VAR_OUTPUT
	Auto: 				BOOL;
	Manual: 			BOOL;
	Faulted: 			BOOL;
//	Sts_StateCntrl:	ST_StateCntrlSts;
END_VAR

VAR
	Warning_ftrig: 		F_TRIG;
	CrntStateold: 		E_StateCntrl;
	sTempLabel: 		STRING;
END_VAR

// Set Up State on Initialization
IF IN_Init THEN
	Sts_StateCntrl.CrntState := CfgDefState;
	(*
		Increment the CFG_EquipIndex
		If the value is different than the currently stored value, update the local index
	*)
	IF Sts_StateCntrl.Index = 0 THEN
		CFG_EquipIndex := CFG_EquipIndex + 1;
		Sts_StateCntrl.Index := CFG_EquipIndex;
	END_IF
	
	//	Test the CFG_EquipLabel for a value
	IF CFG_EquipLabel = '' THEN
		sTempLabel := F_PaddNumber(CFG_EquipIndex, 4, '0',0);
		CFG_EquipLabel := CONCAT('E',sTempLabel);
	END_IF
	// Assign the Equipment Label value to the Status Label item
	Sts_StateCntrl.Label := CFG_EquipLabel;
ELSE
	// Track State Change
	IF Sts_StateCntrl.StateChanged THEN
		Sts_StateCntrl.LstState := CrntStateold;
		CrntStateold := Sts_StateCntrl.CrntState;
		Sts_StateCntrl.StateChanged := FALSE;
	END_IF
	
	//Clear One Scan Received Notices
	IF Sts_StateCntrl.Received.OfflinePB THEN Sts_StateCntrl.Received.OfflinePB := FALSE; END_IF
	IF Sts_StateCntrl.Received.AutoPB THEN Sts_StateCntrl.Received.AutoPB := FALSE; END_IF
	IF Sts_StateCntrl.Received.ManPB THEN Sts_StateCntrl.Received.ManPB := FALSE; END_IF
	IF Sts_StateCntrl.Received.StopPB THEN Sts_StateCntrl.Received.StopPB := FALSE; END_IF
	IF Sts_StateCntrl.Received.ResetPB THEN Sts_StateCntrl.Received.ResetPB := FALSE; END_IF
	IF Sts_StateCntrl.Received.ManMotorRunPB THEN Sts_StateCntrl.Received.ManMotorRunPB := FALSE; END_IF
	IF Sts_StateCntrl.Received.ManExtendPB THEN Sts_StateCntrl.Received.ManExtendPB := FALSE; END_IF
	IF Sts_StateCntrl.Received.ManRetractPB THEN Sts_StateCntrl.Received.ManRetractPB := FALSE; END_IF
	IF Sts_StateCntrl.RcvdFault THEN Sts_StateCntrl.RcvdFault := FALSE; END_IF
	
	
	// Choose logic based on current state
	CASE Sts_StateCntrl.CrntState OF
		//Offline  
		E_StateCntrl.stOffline:
			Sts_StateCntrl.CrntStateTxt := 'Offline';
			Sts_StateCntrl.StateRunOK := FALSE;
			
			IF o_StatePB.ManPB THEN
				Sts_StateCntrl.Received.ManPB := TRUE; 
				Sts_StateCntrl.CrntState := E_StateCntrl.stManual;	
			END_IF
				
		// Auto, transition to manual/faulted are the only allowable state transitions 
		E_StateCntrl.stAuto:
			Sts_StateCntrl.CrntStateTxt := 'Auto';
			IF IN_Fault THEN
				Sts_StateCntrl.RcvdFault := TRUE;
				Sts_StateCntrl.CrntState := E_StateCntrl.stFaulted;
			ELSIF o_StatePB.ManPB 
			   OR p_StatePB.ManPB 
			   OR o_StatePB.StopPB 
			   OR p_StatePB.StopPB 
			   THEN
				IF o_StatePB.ManPB 
				   OR p_StatePB.ManPB
				   THEN
					Sts_StateCntrl.Received.ManPB := TRUE; 
				END_IF
				IF o_StatePB.StopPB 
				   OR p_StatePB.StopPB
				   THEN
					Sts_StateCntrl.Received.StopPB := TRUE; 
				END_IF
				Sts_StateCntrl.StateRunOK := FALSE;
				Sts_StateCntrl.CrntState := E_StateCntrl.stManual;				
			END_IF
			
			IF P_ReqRun AND (Sts_StateCntrl.CrntState = E_StateCntrl.stAuto )THEN
				Sts_StateCntrl.StateRunOK := TRUE;
			ELSE 
				Sts_StateCntrl.StateRunOK := FALSE;
			END_IF
			
		//Manual,transition to auto/offline/faulted are the only allowable state transitions
		E_StateCntrl.stManual:
		Sts_StateCntrl.CrntStateTxt := 'Manual';
			IF IN_Fault THEN
				Sts_StateCntrl.RcvdFault := TRUE;
				Sts_StateCntrl.CrntState := E_StateCntrl.stFaulted;
			ELSIF o_StatePB.OfflinePB OR p_StatePB.OfflinePB THEN
				Sts_StateCntrl.Received.OfflinePB := TRUE; 
				Sts_StateCntrl.CrntState := E_StateCntrl.stOffline;
			ELSIF o_StatePB.AutoPB OR p_StatePB.AutoPB  THEN 
				Sts_StateCntrl.Received.AutoPB := TRUE;
				Sts_StateCntrl.CrntState := E_StateCntrl.stAuto;					
			END_IF
			
			IF o_StatePB.StopPB THEN
				Sts_StateCntrl.Received.StopPB :=TRUE;
				Sts_StateCntrl.StateRunOK := FALSE;
			ELSIF o_StatePB.ManMotorRunPB
			   OR o_StatePB.ManExtendPB
			   OR o_StatePB.ManRetractPB
			   THEN
				// Motor Run
				IF o_StatePB.ManMotorRunPB
				   THEN
						Sts_StateCntrl.Received.ManMotorRunPB := TRUE;
				END_IF
				// Solenoid Extend
				IF o_StatePB.ManExtendPB
				   THEN
						Sts_StateCntrl.Received.ManExtendPB := TRUE;
				END_IF
				// Solenoid Retract
				IF o_StatePB.ManRetractPB
				   THEN
						Sts_StateCntrl.Received.ManRetractPB := TRUE;
				END_IF
				Sts_StateCntrl.StateRunOK := TRUE;
			END_IF
			
		// Faulted - Can initiate a reset or transition to Offline
		E_StateCntrl.stFaulted:
			Sts_StateCntrl.CrntStateTxt := 'Faulted';
			Sts_StateCntrl.StateRunOK := FALSE;
			
			IF o_StatePB.ResetPB OR p_StatePB.ResetPB THEN
				Sts_StateCntrl.Received.ResetPB := TRUE;
				Sts_StateCntrl.CrntState := CfgDefState;
			ELSIF o_StatePB.OfflinePB THEN
				Sts_StateCntrl.Received.ResetPB := TRUE; 
				Sts_StateCntrl.CrntState := E_StateCntrl.stOffline;
			END_IF
	END_CASE
	
			
	// Watch If State Changed
	IF CrntStateold <> Sts_StateCntrl.CrntState AND NOT Sts_StateCntrl.StateChanged THEN
		Sts_StateCntrl.StateChanged := TRUE;
	END_IF
	
	//Show Testing Outputs
	Sts_StateCntrl.StsOffline := Sts_StateCntrl.CrntState = E_StateCntrl.stOffline;
	Sts_StateCntrl.StsAuto := Sts_StateCntrl.CrntState = E_StateCntrl.stAuto;
	Sts_StateCntrl.StsMan := Sts_StateCntrl.CrntState = E_StateCntrl.stManual;
	Sts_StateCntrl.StsFaulted := Sts_StateCntrl.CrntState = E_StateCntrl.stFaulted;
END_IF

END_FUNCTION_BLOCK

// ---- FunctionBlocks/Utils/F_PaddNumber.TcPOU
FUNCTION F_PaddNumber : STRING
VAR_INPUT
	nNumberToConvert: DINT; // Number to convert to string
	nCharsToReturn: DINT;	// Number of Characters to Pad
	sCharToPaddWith: STRING[1] := '0';	// Character to Pad with
	bLeftJustify: BOOL := 0;	// If true, justify to the Left, pad to the right
END_VAR
VAR
	sConvertedString: STRING;	// Number converted to string
	nStringLength: INT;	// Length of the original string
END_VAR

// Convert the number to a string
sConvertedString := TO_STRING(nNumberToConvert);

// Get the length of the converted string
nStringLength := LEN(sConvertedString);

// Test the length to varify it is not longer than the requested length
IF nStringLength < nCharsToReturn THEN
	// Pad the string to length, either to the left or right
	WHILE nStringLength < nCharsToReturn DO
		IF bLeftJustify THEN
			sConvertedString := CONCAT(sConvertedString, sChartoPaddWith);
		else
			sConvertedString := CONCAT(sConvertedString, sChartoPaddWith);
		END_IF
		nStringLength := LEN(sConvertedString);
	END_WHILE
	F_PaddNumber := sConvertedString;
ELSE
	// If the number is longer, just cut it off
	IF bLeftJustify THEN
		F_PaddNumber := LEFT(sConvertedString, TO_INT(nCharsToReturn));
	ELSE
		F_PaddNumber := RIGHT(sConvertedString, TO_INT(nCharsToReturn));
	END_IF
END_IF

END_FUNCTION

// ---- FunctionBlocks/Conveyance/FB_SleepCntrl.TcPOU
(*
Description:
	Function Block to control a sleep timer based on In_CrntMtrFeedBack input, In_TrigArry input and a DisableSleepTmr input.
	Time is configurable with CFG_WaitToSlpTime.
	Timer is reset if any of the triggers are TRUE.
	Timer will run if there is no trigger input and feedback is TRUE. 
	If Timer elapses then the SleepActive output is TRUE until reset by a TRUE in the In_TrigArry
*) 
FUNCTION_BLOCK FB_SleepCntrl
(*
Version history:
 +-------------+------------+----------------+----------+-------------------------------------------+
 |Date         | Version    | created under  | Author   | Remark                                   	|
 +=============+============+================+==========+===========================================+
 |2019-06-11   | 1.0.0.0    | V3.1.0.0       | D.J.     | Initial Release                          	|
 |2019-11-13   | 1.0.0.0    | V3.1.0.0       | D.J.     | Added External Wake trigger              	|
 |2020-02-19   | 1.0.0.0    | V3.1.0.0       | C.Y.     | Changed from array to UINT to trigger		|
 +-------------+------------+----------------+----------+-------------------------------------------+
*)
  
VAR_INPUT
	In_Trigs:	UINT;		// Non-Zero value wakes from sleep 
	In_ExternalTrig: BOOL;		// An external wake trigger	
	In_CrntFeedBack: BOOL;		// The current (Motor or Enable) Feedback (Current feedback 0=Off, 1= Running)
	CFG_WaitToSlpTime:	TIME;		// Time to wait after last trigger before enabling the sleep output
	DisableSleepTmr:	BOOL;		// Input to disable Sleep Timer
	In_ConvState:		E_StateCntrl;	// Detect Auto
END_VAR
VAR_OUTPUT
	SleepActive:	BOOL;		// Sleep is Active Output
END_VAR
VAR
	SleepTimerTon: TON;		// Timer
	ResetTimer: BOOL;		// Internal Flag to reset timer based on input arry
END_VAR

// Set Reset of Timer
ResetTimer := (In_ExternalTrig OR In_Trigs > 0) OR In_ConvState <> E_StateCntrl.stAuto;

// Timer Call
SleepTimerTon(IN:= In_CrntFeedBack AND (NOT ResetTimer) AND (NOT DisableSleepTmr) , PT:= CFG_WaitToSlpTime, Q=> );

// Set Output
IF SleepTimerTon.Q THEN
	SleepActive := TRUE;
ELSIF ResetTimer THEN
	SleepActive := FALSE;
END_IF;

END_FUNCTION_BLOCK

// ---- FunctionBlocks/VFD/Functions/VFD.TcPOU
FUNCTION_BLOCK VFD
FUNCTION_BLOCK VFD
VAR_INPUT
	RunVelocity				: INT;
	RunRequest				: BOOL;
	PLCFault				: BOOL;
	Reset					: BOOL;
	VelocityThreshold		: INT;
END_VAR
VAR_OUTPUT
	ActualVelocity 	AT %I* 	: INT;
	StatusWord		AT %I* 	: UINT;
	Run_OK					: BOOL;
	STO_Active				: BOOL;
	IsRunning				: BOOL;
	IsFaulted 				: BOOL;
END_VAR
VAR
	VFD_State				: DriveState;
	ControlWord 	AT %Q* 	: UINT;
	TargetVelocity 	AT %Q*	: INT;
	StatusWordFiltered		: UINT;
END_VAR
VAR CONSTANT
	SAFETY_TORQUE_OFF_ACTIVE : INT := 15;
END_VAR

StatusWordFiltered := StatusWord AND 16#006F;

VFD_State(StatusWord := StatusWordFiltered, Run_Drive := RunRequest, ControlWord => ControlWord, PLCFault := PLCFault, ResetFault := Reset);

IF Reset THEN
	Reset := FALSE;
END_IF

Run_OK := (StatusWordFiltered = Drive_State.READY_TO_SWITCH_ON) OR (StatusWordFiltered = Drive_State.SWITCHED_ON) OR (StatusWordFiltered = Drive_State.OPERATION_ENABLED);

IF StatusWordFiltered = Drive_State.OPERATION_ENABLED THEN
	TargetVelocity := RunVelocity;
ELSE
	TargetVelocity := 0;	
END_IF

STO_Active := StatusWord.SAFETY_TORQUE_OFF_ACTIVE;
 
IsRunning := ActualVelocity >= VelocityThreshold;
IsFaulted := VFD_State.Fault;

END_FUNCTION_BLOCK

// ---- FunctionBlocks/VFD/Functions/DriveState.TcPOU
FUNCTION_BLOCK DriveState
VAR_INPUT
	StatusWord : UINT;
	PLCFault   : BOOL;
	ResetFault : BOOL;
	Run_Drive  : BOOL;
END_VAR
VAR_OUTPUT
	ControlWord : UINT;
	Fault	: BOOL;	
END_VAR
VAR
END_VAR
VAR CONSTANT 
	//Status Word Bit Definitions
	READY_TO_SWITCH_ON 	: INT := 0;
	SWITCHED_ON			: INT := 1;
	OPERATION_ENABLED	: INT := 2;
	FAULT_ACTIVE		: INT := 3;
	DC_BUS_READY		: INT := 4;
	QUICK_STOP_INACTIVE	: INT := 5;
	OPERATION_INHIBITED : INT := 6;
	WARNING_ACTIVE		: INT := 7;
	
	//Control Word Bit Definitions
	SWITCH_ON			: INT := 0;
	ESTABLISH_READINESS	: INT := 1;
	ACTIVATE_QUICK_STOP	: INT := 2;
	OPERATION_ENABLE 	: INT := 3;
	RAMP_OUT_ZERO		: INT := 4;
	RAMP_HOLD			: INT := 5;
	RAMP_IN_ZERO		: INT := 6;
	
	//Bits 4-6 are operating mode dependent and not supported with CiA402 profile
	RESET_FAULT			: INT := 7;
END_VAR


CASE StatusWord OF
	
	DRIVE_STATE.NOT_READY_TO_SWITCH_ON, DRIVE_STATE.NOT_READY_TO_SWITCH_ON_BIT_5: 
		//No Control word is needed here because drive will automatically advance as long as it has been initialized properly
		
	DRIVE_STATE.SWITCH_ON_INHIBITED, DRIVE_STATE.SWITCH_ON_INHIBITED_BIT_5:	
		
		FAULT := FALSE;
		//GO TO READY TO SWITCH ON
		ControlWord.SWITCH_ON := 0;
		ControlWord.ESTABLISH_READINESS := 1;
		ControlWord.ACTIVATE_QUICK_STOP := 1;
		ControlWord.RESET_FAULT			:= 0;
	
	DRIVE_STATE.READY_TO_SWITCH_ON:
		
		IF NOT StatusWord.QUICK_STOP_INACTIVE THEN 
			//GO TO SWITCH ON INHIBITED
			ControlWord.ESTABLISH_READINESS := 1;
			ControlWord.ACTIVATE_QUICK_STOP := 0;
			ControlWord.RESET_FAULT			:= 0;
		ELSIF Run_Drive THEN 
			//GO TO SWITCHED ON
			ControlWord.SWITCH_ON := 1;
			ControlWord.ESTABLISH_READINESS := 1;
			ControlWord.ACTIVATE_QUICK_STOP := 1;
			ControlWord.OPERATION_ENABLE	:= 0;
			ControlWord.RESET_FAULT			:= 0;
			ControlWord.RAMP_OUT_ZERO		:= 1;
			ControlWord.RAMP_HOLD			:= 1;
			ControlWord.RAMP_IN_ZERO		:= 1;
		ELSIF PLCFault THEN
			//GO TO SWITCH ON INHIBITED
			ControlWord.ESTABLISH_READINESS := 0;
			ControlWord.RESET_FAULT			:= 0;
		END_IF
	
	DRIVE_STATE.SWITCHED_ON:
	
		IF NOT StatusWord.QUICK_STOP_INACTIVE THEN
			//GO TO SWITCH ON INHIBITED
			ControlWord.ESTABLISH_READINESS := 1;
			ControlWord.ACTIVATE_QUICK_STOP := 0;
			ControlWord.RESET_FAULT			:= 0;
		ELSIF RUN_DRIVE THEN
			//GO TO OPERATION ENABLED
			ControlWord.SWITCH_ON := 1;
			ControlWord.ESTABLISH_READINESS := 1;
			ControlWord.ACTIVATE_QUICK_STOP := 1;
			ControlWord.OPERATION_ENABLE	:= 1;
			ControlWord.RESET_FAULT			:= 0;
		ELSE
			//GO TO READY TO SWITCH ON
			ControlWord.SWITCH_ON := 0;
			ControlWord.ESTABLISH_READINESS := 1;
			ControlWord.ACTIVATE_QUICK_STOP := 1;
			ControlWord.RESET_FAULT			:= 0;
		END_IF

	DRIVE_STATE.OPERATION_ENABLED:
		
		IF (NOT StatusWord.QUICK_STOP_INACTIVE) THEN
			//GO TO QUICK STOP ACTIVE
			ControlWord.ESTABLISH_READINESS := 1;
			ControlWord.ACTIVATE_QUICK_STOP := 0;
			ControlWord.RESET_FAULT			:= 0;
						
		ELSIF NOT Run_Drive THEN
			//GO TO SWITCHED ON
			ControlWord.SWITCH_ON := 1;
			ControlWord.ESTABLISH_READINESS := 1;
			ControlWord.ACTIVATE_QUICK_STOP := 1;
			ControlWord.OPERATION_ENABLE	:= 0;
			ControlWord.RESET_FAULT			:= 0;
			ControlWord.RAMP_OUT_ZERO		:= 0;
			ControlWord.RAMP_HOLD			:= 0;
			ControlWord.RAMP_IN_ZERO		:= 0;
		END_IF
		
	DRIVE_STATE.QUICK_STOP_ACTIVE:

		IF Run_Drive THEN
			//GO TO OPERATION ENABLED
			ControlWord.SWITCH_ON := 1;
			ControlWord.ESTABLISH_READINESS := 1;
			ControlWord.ACTIVATE_QUICK_STOP := 1;
			ControlWord.OPERATION_ENABLE	:= 1;
			ControlWord.RESET_FAULT			:= 0;
		ELSE
			//GO TO SWITCH ON INHIBITED
			ControlWord.ESTABLISH_READINESS := 0;
			ControlWord.RESET_FAULT			:= 0;
		END_IF	
		
	DRIVE_STATE.TROUBLE, DRIVE_STATE.TROUBLE_BIT_5, DRIVE_STATE.FAULT_REACTION_ACTIVE, DRIVE_STATE.FAULT_REACTION_ACTIVE_BIT_5:	
	
		FAULT := TRUE;
			
		IF ControlWord <> 16#0000 THEN
			ControlWord := 16#0000;
		ELSIF ResetFault THEN
			ControlWord := 16#0080;
		END_IF;			
END_CASE

END_FUNCTION_BLOCK

// ---- POUs/CommStatus.TcPOU
PROGRAM CommStatus
VAR
	DebounceOnTime:	TIME := T#500MS;     // Default Value	
	DebounceOffTime:	TIME := T#1S;     // Default Value
		
	RIO1151_CommFault: FB_DigDebnce;	// Remote IO Block 1151 Communication Fault
	RIO2151_CommFault: FB_DigDebnce;	// Remote IO Block 2151 Communication Fault
	RIO3171_CommFault: FB_DigDebnce;	// Remote IO Block 3171 Communication Fault
	RIO4141_CommFault: FB_DigDebnce;	// Remote IO Block 4141 Communication Fault
	RIO7151_CommFault: FB_DigDebnce;	// Remote IO Block 7151 Communication Fault
	RIO8171_CommFault: FB_DigDebnce;	// Remote IO Block 8171 Communication Fault
	RIO9191_CommFault: FB_DigDebnce;	// Remote IO Block 9191 Communication Fault
	RIO10161_CommFault: FB_DigDebnce;	// Remote IO Block 10161 Communication Fault
	RIO11171_CommFault: FB_DigDebnce;	// Remote IO Block 11171 Communication Fault
	RIO12182_CommFault: FB_DigDebnce;	// Remote IO Block 12182 Communication Fault
	
	BCR_S2140_01_CommFault: FB_DigDebnce;;		// Bar Code Reader 2140_01 Communication Fault
	BCR_S2141_01_CommFault: FB_DigDebnce;;		// Bar Code Reader 2141_01 Communication Fault
	BCR_S2150_01_CommFault: FB_DigDebnce;;		// Bar Code Reader 2150_01 Communication Fault
	BCR_S3080_01_CommFault: FB_DigDebnce;;		// Bar Code Reader 3080_01 Communication Fault
	
	Ethernet_CommFault: FB_DigDebnce;;		// Ethernet Adapter Status Communication Fault
	
END_VAR

// Remote IO Blocks --------------------
RIO1151_CommFault(
	In:= GVL_IO.RIO1151_WcState, 
	CFG_OKState:= 0, 
	CFG_OnDlyTime:= DebounceOnTime, 
	CFG_OffDlyTime:= DebounceOffTime, 
	In_Sim:= , 
	);

RIO2151_CommFault(
	In:= GVL_IO.RIO2151_WcState, 
	CFG_OKState:= 0, 
	CFG_OnDlyTime:= DebounceOnTime, 
	CFG_OffDlyTime:= DebounceOffTime, 
	In_Sim:= , 
	);
	
RIO3171_CommFault(
	In:= GVL_IO.RIO3171_WcState, 
	CFG_OKState:= 0, 
	CFG_OnDlyTime:= DebounceOnTime, 
	CFG_OffDlyTime:= DebounceOffTime, 
	In_Sim:= , 
	);
	
RIO4141_CommFault(
	In:= GVL_IO.RIO4141_WcState, 
	CFG_OKState:= 0, 
	CFG_OnDlyTime:= DebounceOnTime, 
	CFG_OffDlyTime:= DebounceOffTime, 
	In_Sim:= , 
	);
	
RIO7151_CommFault(
	In:= GVL_IO.RIO7151_WcState, 
	CFG_OKState:= 0, 
	CFG_OnDlyTime:= DebounceOnTime, 
	CFG_OffDlyTime:= DebounceOffTime, 
	In_Sim:= , 
	);
	
RIO8171_CommFault(
	In:= GVL_IO.RIO8171_WcState, 
	CFG_OKState:= 0, 
	CFG_OnDlyTime:= DebounceOnTime, 
	CFG_OffDlyTime:= DebounceOffTime, 
	In_Sim:= , 
	);
	
RIO9191_CommFault(
	In:= GVL_IO.RIO9191_WcState, 
	CFG_OKState:= 0, 
	CFG_OnDlyTime:= DebounceOnTime, 
	CFG_OffDlyTime:= DebounceOffTime, 
	In_Sim:= , 
	);
	
RIO10161_CommFault(
	In:= GVL_IO.RIO10161_WcState, 
	CFG_OKState:= 0, 
	CFG_OnDlyTime:= DebounceOnTime, 
	CFG_OffDlyTime:= DebounceOffTime, 
	In_Sim:= , 
	);
	
RIO11171_CommFault(
	In:= GVL_IO.RIO11171_WcState, 
	CFG_OKState:= 0, 
	CFG_OnDlyTime:= DebounceOnTime, 
	CFG_OffDlyTime:= DebounceOffTime, 
	In_Sim:= , 
	);

RIO12182_CommFault(
	In:= GVL_IO.RIO12182_WcState , 
	CFG_OKState:= 0, 
	CFG_OnDlyTime:= DebounceOnTime, 
	CFG_OffDlyTime:= DebounceOffTime, 
	In_Sim:= , 
	);

// Bar Code Readers --------------------	
BCR_S2140_01_CommFault(
	In:= BarCodeReaders.BCR_S2140_01.Out_DeviceState = 0, 
	CFG_OKState:= 1, 
	CFG_OnDlyTime:= DebounceOnTime, 
	CFG_OffDlyTime:= DebounceOffTime, 
	In_Sim:= , 
	);
	
BCR_S2141_01_CommFault(
	In:= BarCodeReaders.BCR_S2141_01.Out_DeviceState = 0, 
	CFG_OKState:= 1, 
	CFG_OnDlyTime:= DebounceOnTime, 
	CFG_OffDlyTime:= DebounceOffTime, 
	In_Sim:= , 
	);
	
BCR_S2150_01_CommFault(
	In:= BarCodeReaders.BCR_S2150_01.Out_DeviceState = 0, 
	CFG_OKState:= 1, 
	CFG_OnDlyTime:= DebounceOnTime, 
	CFG_OffDlyTime:= DebounceOffTime, 
	In_Sim:= , 
	);
	
BCR_S3080_01_CommFault(
	In:= BarCodeReaders.BCR_S3080_01.Out_DeviceState = 0, 
	CFG_OKState:= 1, 
	CFG_OnDlyTime:= DebounceOnTime, 
	CFG_OffDlyTime:= DebounceOffTime, 
	In_Sim:= , 
	);
	
// Ethernet Controller	
Ethernet_CommFault(
//	In:= GVL_IO.EthernetAdapter_State = 0, 
	CFG_OKState:= 1, 
	CFG_OnDlyTime:= DebounceOnTime, 
	CFG_OffDlyTime:= DebounceOffTime, 
	In_Sim:= , 
	);

END_PROGRAM

// ---- POUs/ProxSensors.TcPOU
PROGRAM ProxSensors
VAR
DebounceOnTime:	TIME := T#5MS;     // Default Value
DebounceOffTime:	TIME := T#500MS;     // Default Value
JamDetectTime:	TIME := T#5S;     // Default Value

In_PX_2131_Extended AT %I* : BOOL;      // Mapped IO input for PX
PX_2131_Extended:  FB_DigDebnce;		// PI2150-01 PIN STOP EXTENDED PROX

In_PX_2151_Retracted AT %I* : BOOL;      // Mapped IO input for PX
PX_2151_Retracted:  FB_DigDebnce;		// PI2150-01 PIN STOP GRIPPER RETRACTED PROX

In_PX_2181_Extended AT %I* : BOOL;      // Mapped IO input for PX
PX_2181_Extended:  FB_DigDebnce;		// GR2150-01 "BELT" GRIPPER EXTENDED PROX

In_PX_2201_Retracted AT %I* : BOOL;      // Mapped IO input for PX
PX_2201_Retracted:  FB_DigDebnce;		// GR2150-01 "BELT" GRIPPER RETRACTED PROX

In_PX_3171_Extended AT %I* : BOOL;      // Mapped IO input for PX
PX_3171_Extended:  FB_DigDebnce;		// PU2150-02 PUSH DIVERT EXTENDED PROX

In_PX_3191_Retracted AT %I* : BOOL;      // Mapped IO input for PX
PX_3191_Retracted:  FB_DigDebnce;		// PU2150-02 PUSH DIVERT RETRACTED PROX

In_PX_3301_Extended AT %I* : BOOL;      // Mapped IO input for PX
PX_3301_Extended:  FB_DigDebnce;		// PU2150-01 PUSH DIVERT EXTENDED PROX

In_PX_3331_Retracted AT %I* : BOOL;      // Mapped IO input for PX
PX_3331_Retracted:  FB_DigDebnce;		// PU2150-01 PUSH DIVERT RETRACTED PROX

In_PX_4151_Extended AT %I* : BOOL;      // Mapped IO input for PX
PX_4151_Extended:  FB_DigDebnce;		// PU2150-04 PUSH DIVERT EXTENDED PROX

In_PX_4171_Retracted AT %I* : BOOL;      // Mapped IO input for PX
PX_4171_Retracted:  FB_DigDebnce;		// PU2150-04 PUSH DIVERT RETRACTED PROX

In_PX_4291_Extended AT %I* : BOOL;      // Mapped IO input for PX
PX_4291_Extended:  FB_DigDebnce;		// PU2150-03 PUSH DIVERT EXTENDED PROX

In_PX_4311_Retracted AT %I* : BOOL;      // Mapped IO input for PX
PX_4311_Retracted:  FB_DigDebnce;		// PU2150-03 PUSH DIVERT RETRACTED PROX

In_PX_10181_Extended AT %I* : BOOL;      // Mapped IO input for PX
PX_10181_Extended:  FB_DigDebnce;		// PL2140 PLOW DIVERT PISTON PROX EXTENDED PROX

In_PX_10211_Extended AT %I* : BOOL;      // Mapped IO input for PX
PX_10211_Extended:  FB_DigDebnce;		// PL2140 PLOW DIVERT EXTENDED PROX

In_PX_10231_Retracted AT %I* : BOOL;      // Mapped IO input for PX
PX_10231_Retracted:  FB_DigDebnce;		// PL2140 PLOW DIVERT RETRACTED PROX

In_PX_11181_Extended AT %I* : BOOL;      // Mapped IO input for PX
PX_11181_Extended:  FB_DigDebnce;		// PI2140 PIN STOP EXTENDED PROX

In_PX_11201_Retracted AT %I* : BOOL;      // Mapped IO input for PX
PX_11201_Retracted:  FB_DigDebnce;		// PI2140 PIN STOP RETRACTED PROX

In_PX_11291_Extended AT %I* : BOOL;      // Mapped IO input for PX
PX_11291_Extended:  FB_DigDebnce;		// GR2140-02 "D" GRIPPER EXTENDED PROX

In_PX_11321_Retracted AT %I* : BOOL;      // Mapped IO input for PX
PX_11321_Retracted:  FB_DigDebnce;		// GR2140-02 "D" GRIPPER RETRACTED PROX

In_PX_11141_Extended AT %I* : BOOL;      // Mapped IO input for PX
PX_11141_Extended:  FB_DigDebnce;		// GR2140-01 "D" GRIPPER EXTENDED PROX

In_PX_11161_Retracted AT %I* : BOOL;      // Mapped IO input for PX
PX_11161_Retracted:  FB_DigDebnce;		// GR2140-01 "D" GRIPPER RETRACTED PROX

In_PX_12151_Extended AT %I* : BOOL;      // Mapped IO input for PX
PX_12151_Extended:  FB_DigDebnce;		// P2130 PROX BREAK AWAY EXTENDED PROX

In_PX_12251_Extended AT %I* : BOOL;      // Mapped IO input for PX
PX_12251_Extended:  FB_DigDebnce;		// P3095 PROX BREAK AWAY EXTENDED PROX
END_VAR

// PI2150-01 PIN STOP GRIPPER Extended
PX_2131_Extended(
	In:= In_PX_2131_Extended,
	CFG_OKState:= 0,
	CFG_OnDlyTime:= DebounceOnTime,
	CFG_OnDlyTime:= DebounceOffTime,
	In_Sim:= 
	);

// PI2150-01 PIN STOP GRIPPER Retracted
PX_2151_Retracted(
	In:= In_PX_2151_Retracted,
	CFG_OKState:= 0,
	CFG_OnDlyTime:= DebounceOnTime,
	CFG_OnDlyTime:= DebounceOffTime,
	In_Sim:= 
	);

// GR2150-01 "BELT" GRIPPER Extended
PX_2181_Extended(
	In:= In_PX_2181_Extended,
	CFG_OKState:= 0,
	CFG_OnDlyTime:= DebounceOnTime,
	CFG_OnDlyTime:= DebounceOffTime,
	In_Sim:= 
	);

// GR2150-01 "BELT" GRIPPER Retracted
PX_2201_Retracted(
	In:= In_PX_2201_Retracted,
	CFG_OKState:= 0,
	CFG_OnDlyTime:= DebounceOnTime,
	CFG_OnDlyTime:= DebounceOffTime,
	In_Sim:= 
	);

// PU2150-02 PUSH DIVERT Extended
PX_3171_Extended(
	In:= In_PX_3171_Extended,
	CFG_OKState:= 0,
	CFG_OnDlyTime:= DebounceOnTime,
	CFG_OnDlyTime:= DebounceOffTime,
	In_Sim:= 
	);

// PU2150-02 PUSH DIVERT Retracted
PX_3191_Retracted(
	In:= In_PX_3191_Retracted,
	CFG_OKState:= 0,
	CFG_OnDlyTime:= DebounceOnTime,
	CFG_OnDlyTime:= DebounceOffTime,
	In_Sim:= 
	);

// PU2150-01 PUSH DIVERT Extended
PX_3301_Extended(
	In:= In_PX_3301_Extended,
	CFG_OKState:= 0,
	CFG_OnDlyTime:= DebounceOnTime,
	CFG_OnDlyTime:= DebounceOffTime,
	In_Sim:= 
	);

// PU2150-01 PUSH DIVERT Retracted
PX_3331_Retracted(
	In:= In_PX_3331_Retracted,
	CFG_OKState:= 0,
	CFG_OnDlyTime:= DebounceOnTime,
	CFG_OnDlyTime:= DebounceOffTime,
	In_Sim:= 
	);

// PU2150-04 PUSH DIVERT Extended
PX_4151_Extended(
	In:= In_PX_4151_Extended,
	CFG_OKState:= 0,
	CFG_OnDlyTime:= DebounceOnTime,
	CFG_OnDlyTime:= DebounceOffTime,
	In_Sim:= 
	);

// PU2150-04 PUSH DIVERT Retracted
PX_4171_Retracted(
	In:= In_PX_4171_Retracted,
	CFG_OKState:= 0,
	CFG_OnDlyTime:= DebounceOnTime,
	CFG_OnDlyTime:= DebounceOffTime,
	In_Sim:= 
	);

